;FOLD ARCOFF WDAT2 LIN P4 CPDAT2 Tool[1]:cmttorch Base[1]:vrashatel ;%{PE}
  ;FOLD Parameters ;%{h}
    ;Params IlfProvider=kukaroboter.arctech.arcofflin; Kuka.IsGlobalPoint=False; Kuka.PointName=P4; Kuka.BlendingEnabled=False; Kuka.MoveDataName=CPDAT2; Kuka.VelocityPath=0.01; Kuka.CurrentCDSetIndex=0; Kuka.MovementParameterFieldEnabled=True; ArcTech.WdatVarName=WDAT2; ArcTech.Basic=3.4.3.1264
  ;ENDFOLD
  $BWDSTART = FALSE
  LDAT_ACT = LCPDAT2
  FDAT_ACT = FP4
  BAS(#CP_PARAMS, gArcBasVelDefinition)
  SET_CD_PARAMS (0)
  TRIGGER WHEN PATH = ArcGetPath(#ArcOffBefore, WDAT2) DELAY = 0 DO ArcMainNG(#ArcOffBeforeOffStd, WDAT2, WP4) PRIO = -1
  TRIGGER WHEN PATH = ArcGetPath(#OnTheFlyArcOff, WDAT2) DELAY = 0 DO ArcMainNG(#ArcOffMoveStd, WDAT2, WP4) PRIO = -1
  ArcMainNG(#ArcOffBeforeMoveStd, WDAT2, WP4)
  LIN XP4
  ArcMainNG(#ArcOffAfterMoveStd, WDAT2, WP4)
;ENDFOLD
   $VEL.CP = 0.080
   LIN  {X 8.829, Y -0.910, Z 19.700, A 0.000, B 0.000, C 0.000} C_DIS

;FOLD ARCON WDAT1 LIN P3 Vel=0.5 m/s CPDAT1 Tool[1]:cmttorch Base[1]:vrashatel ;%{PE}
  ;FOLD Parameters ;%{h}
    ;Params IlfProvider=kukaroboter.arctech.arconlin; Kuka.IsGlobalPoint=False; Kuka.PointName=P3; Kuka.BlendingEnabled=False; Kuka.MoveDataName=CPDAT1; Kuka.VelocityPath=0.5; Kuka.CurrentCDSetIndex=0; Kuka.MovementParameterFieldEnabled=True; ArcTech.WdatVarName=WDAT1; ArcTech.Basic=3.4.3.1264
  ;ENDFOLD
  $BWDSTART = FALSE
  LDAT_ACT = LCPDAT1
  FDAT_ACT = FP3
  BAS(#CP_PARAMS, 0.5)
  SET_CD_PARAMS (0)
  TRIGGER WHEN DISTANCE = 1 DELAY = ArcGetDelay(#PreDefinition, WDAT1) DO ArcMainNG(#PreDefinition, WDAT1, WP3) PRIO = -1
  TRIGGER WHEN PATH = ArcGetPath(#OnTheFlyArcOn, WDAT1) DELAY = ArcGetDelay(#GasPreflow, WDAT1) DO ArcMainNG(#GasPreflow, WDAT1, WP3) PRIO = -1
  TRIGGER WHEN PATH = ArcGetPath(#OnTheFlyArcOn, WDAT1) DELAY = 0 DO ArcMainNG(#ArcOnMoveStd, WDAT1, WP3) PRIO = -1
  ArcMainNG(#ArcOnBeforeMoveStd, WDAT1, WP3)
  LIN XP3
  ArcMainNG(#ArcOnAfterMoveStd, WDAT1, WP3)
;ENDFOLD
   $VEL.CP = 0.060
   LIN  {X 4.151, Y 3.768, Z 19.700, A 0.000, B 0.000, C 0.000} C_DIS

;FOLD ARCOFF WDAT2 LIN P4 CPDAT2 Tool[1]:cmttorch Base[1]:vrashatel ;%{PE}
  ;FOLD Parameters ;%{h}
    ;Params IlfProvider=kukaroboter.arctech.arcofflin; Kuka.IsGlobalPoint=False; Kuka.PointName=P4; Kuka.BlendingEnabled=False; Kuka.MoveDataName=CPDAT2; Kuka.VelocityPath=0.01; Kuka.CurrentCDSetIndex=0; Kuka.MovementParameterFieldEnabled=True; ArcTech.WdatVarName=WDAT2; ArcTech.Basic=3.4.3.1264
  ;ENDFOLD
  $BWDSTART = FALSE
  LDAT_ACT = LCPDAT2
  FDAT_ACT = FP4
  BAS(#CP_PARAMS, gArcBasVelDefinition)
  SET_CD_PARAMS (0)
  TRIGGER WHEN PATH = ArcGetPath(#ArcOffBefore, WDAT2) DELAY = 0 DO ArcMainNG(#ArcOffBeforeOffStd, WDAT2, WP4) PRIO = -1
  TRIGGER WHEN PATH = ArcGetPath(#OnTheFlyArcOff, WDAT2) DELAY = 0 DO ArcMainNG(#ArcOffMoveStd, WDAT2, WP4) PRIO = -1
  ArcMainNG(#ArcOffBeforeMoveStd, WDAT2, WP4)
  LIN XP4
  ArcMainNG(#ArcOffAfterMoveStd, WDAT2, WP4)
;ENDFOLD
   $VEL.CP = 0.080
   LIN  {X 4.343, Y 4.142, Z 19.700, A 0.000, B 0.000, C 0.000} C_DIS

;FOLD ARCON WDAT1 LIN P3 Vel=0.5 m/s CPDAT1 Tool[1]:cmttorch Base[1]:vrashatel ;%{PE}
  ;FOLD Parameters ;%{h}
    ;Params IlfProvider=kukaroboter.arctech.arconlin; Kuka.IsGlobalPoint=False; Kuka.PointName=P3; Kuka.BlendingEnabled=False; Kuka.MoveDataName=CPDAT1; Kuka.VelocityPath=0.5; Kuka.CurrentCDSetIndex=0; Kuka.MovementParameterFieldEnabled=True; ArcTech.WdatVarName=WDAT1; ArcTech.Basic=3.4.3.1264
  ;ENDFOLD
  $BWDSTART = FALSE
  LDAT_ACT = LCPDAT1
  FDAT_ACT = FP3
  BAS(#CP_PARAMS, 0.5)
  SET_CD_PARAMS (0)
  TRIGGER WHEN DISTANCE = 1 DELAY = ArcGetDelay(#PreDefinition, WDAT1) DO ArcMainNG(#PreDefinition, WDAT1, WP3) PRIO = -1
  TRIGGER WHEN PATH = ArcGetPath(#OnTheFlyArcOn, WDAT1) DELAY = ArcGetDelay(#GasPreflow, WDAT1) DO ArcMainNG(#GasPreflow, WDAT1, WP3) PRIO = -1
  TRIGGER WHEN PATH = ArcGetPath(#OnTheFlyArcOn, WDAT1) DELAY = 0 DO ArcMainNG(#ArcOnMoveStd, WDAT1, WP3) PRIO = -1
  ArcMainNG(#ArcOnBeforeMoveStd, WDAT1, WP3)
  LIN XP3
  ArcMainNG(#ArcOnAfterMoveStd, WDAT1, WP3)
;ENDFOLD
   $VEL.CP = 0.060
   LIN  {X 8.829, Y -0.344, Z 19.700, A 0.000, B 0.000, C 0.000} C_DIS

;FOLD ARCOFF WDAT2 LIN P4 CPDAT2 Tool[1]:cmttorch Base[1]:vrashatel ;%{PE}
  ;FOLD Parameters ;%{h}
    ;Params IlfProvider=kukaroboter.arctech.arcofflin; Kuka.IsGlobalPoint=False; Kuka.PointName=P4; Kuka.BlendingEnabled=False; Kuka.MoveDataName=CPDAT2; Kuka.VelocityPath=0.01; Kuka.CurrentCDSetIndex=0; Kuka.MovementParameterFieldEnabled=True; ArcTech.WdatVarName=WDAT2; ArcTech.Basic=3.4.3.1264
  ;ENDFOLD
  $BWDSTART = FALSE
  LDAT_ACT = LCPDAT2
  FDAT_ACT = FP4
  BAS(#CP_PARAMS, gArcBasVelDefinition)
  SET_CD_PARAMS (0)
  TRIGGER WHEN PATH = ArcGetPath(#ArcOffBefore, WDAT2) DELAY = 0 DO ArcMainNG(#ArcOffBeforeOffStd, WDAT2, WP4) PRIO = -1
  TRIGGER WHEN PATH = ArcGetPath(#OnTheFlyArcOff, WDAT2) DELAY = 0 DO ArcMainNG(#ArcOffMoveStd, WDAT2, WP4) PRIO = -1
  ArcMainNG(#ArcOffBeforeMoveStd, WDAT2, WP4)
  LIN XP4
  ArcMainNG(#ArcOffAfterMoveStd, WDAT2, WP4)
;ENDFOLD
   $VEL.CP = 0.080
   LIN  {X 8.829, Y 0.221, Z 19.700, A 0.000, B 0.000, C 0.000} C_DIS

;FOLD ARCON WDAT1 LIN P3 Vel=0.5 m/s CPDAT1 Tool[1]:cmttorch Base[1]:vrashatel ;%{PE}
  ;FOLD Parameters ;%{h}
    ;Params IlfProvider=kukaroboter.arctech.arconlin; Kuka.IsGlobalPoint=False; Kuka.PointName=P3; Kuka.BlendingEnabled=False; Kuka.MoveDataName=CPDAT1; Kuka.VelocityPath=0.5; Kuka.CurrentCDSetIndex=0; Kuka.MovementParameterFieldEnabled=True; ArcTech.WdatVarName=WDAT1; ArcTech.Basic=3.4.3.1264
  ;ENDFOLD
  $BWDSTART = FALSE
  LDAT_ACT = LCPDAT1
  FDAT_ACT = FP3
  BAS(#CP_PARAMS, 0.5)
  SET_CD_PARAMS (0)
  TRIGGER WHEN DISTANCE = 1 DELAY = ArcGetDelay(#PreDefinition, WDAT1) DO ArcMainNG(#PreDefinition, WDAT1, WP3) PRIO = -1
  TRIGGER WHEN PATH = ArcGetPath(#OnTheFlyArcOn, WDAT1) DELAY = ArcGetDelay(#GasPreflow, WDAT1) DO ArcMainNG(#GasPreflow, WDAT1, WP3) PRIO = -1
  TRIGGER WHEN PATH = ArcGetPath(#OnTheFlyArcOn, WDAT1) DELAY = 0 DO ArcMainNG(#ArcOnMoveStd, WDAT1, WP3) PRIO = -1
  ArcMainNG(#ArcOnBeforeMoveStd, WDAT1, WP3)
  LIN XP3
  ArcMainNG(#ArcOnAfterMoveStd, WDAT1, WP3)
;ENDFOLD
   $VEL.CP = 0.060
   LIN  {X 4.534, Y 4.516, Z 19.700, A 0.000, B 0.000, C 0.000} C_DIS

;FOLD ARCOFF WDAT2 LIN P4 CPDAT2 Tool[1]:cmttorch Base[1]:vrashatel ;%{PE}
  ;FOLD Parameters ;%{h}
    ;Params IlfProvider=kukaroboter.arctech.arcofflin; Kuka.IsGlobalPoint=False; Kuka.PointName=P4; Kuka.BlendingEnabled=False; Kuka.MoveDataName=CPDAT2; Kuka.VelocityPath=0.01; Kuka.CurrentCDSetIndex=0; Kuka.MovementParameterFieldEnabled=True; ArcTech.WdatVarName=WDAT2; ArcTech.Basic=3.4.3.1264
  ;ENDFOLD
  $BWDSTART = FALSE
  LDAT_ACT = LCPDAT2
  FDAT_ACT = FP4
  BAS(#CP_PARAMS, gArcBasVelDefinition)
  SET_CD_PARAMS (0)
  TRIGGER WHEN PATH = ArcGetPath(#ArcOffBefore, WDAT2) DELAY = 0 DO ArcMainNG(#ArcOffBeforeOffStd, WDAT2, WP4) PRIO = -1
  TRIGGER WHEN PATH = ArcGetPath(#OnTheFlyArcOff, WDAT2) DELAY = 0 DO ArcMainNG(#ArcOffMoveStd, WDAT2, WP4) PRIO = -1
  ArcMainNG(#ArcOffBeforeMoveStd, WDAT2, WP4)
  LIN XP4
  ArcMainNG(#ArcOffAfterMoveStd, WDAT2, WP4)
;ENDFOLD
   $VEL.CP = 0.080
   LIN  {X 4.726, Y 4.890, Z 19.700, A 0.000, B 0.000, C 0.000} C_DIS

;FOLD ARCON WDAT1 LIN P3 Vel=0.5 m/s CPDAT1 Tool[1]:cmttorch Base[1]:vrashatel ;%{PE}
  ;FOLD Parameters ;%{h}
    ;Params IlfProvider=kukaroboter.arctech.arconlin; Kuka.IsGlobalPoint=False; Kuka.PointName=P3; Kuka.BlendingEnabled=False; Kuka.MoveDataName=CPDAT1; Kuka.VelocityPath=0.5; Kuka.CurrentCDSetIndex=0; Kuka.MovementParameterFieldEnabled=True; ArcTech.WdatVarName=WDAT1; ArcTech.Basic=3.4.3.1264
  ;ENDFOLD
  $BWDSTART = FALSE
  LDAT_ACT = LCPDAT1
  FDAT_ACT = FP3
  BAS(#CP_PARAMS, 0.5)
  SET_CD_PARAMS (0)
  TRIGGER WHEN DISTANCE = 1 DELAY = ArcGetDelay(#PreDefinition, WDAT1) DO ArcMainNG(#PreDefinition, WDAT1, WP3) PRIO = -1
  TRIGGER WHEN PATH = ArcGetPath(#OnTheFlyArcOn, WDAT1) DELAY = ArcGetDelay(#GasPreflow, WDAT1) DO ArcMainNG(#GasPreflow, WDAT1, WP3) PRIO = -1
  TRIGGER WHEN PATH = ArcGetPath(#OnTheFlyArcOn, WDAT1) DELAY = 0 DO ArcMainNG(#ArcOnMoveStd, WDAT1, WP3) PRIO = -1
  ArcMainNG(#ArcOnBeforeMoveStd, WDAT1, WP3)
  LIN XP3
  ArcMainNG(#ArcOnAfterMoveStd, WDAT1, WP3)
;ENDFOLD
   $VEL.CP = 0.060
   LIN  {X 8.829, Y 0.787, Z 19.700, A 0.000, B 0.000, C 0.000} C_DIS

;FOLD ARCOFF WDAT2 LIN P4 CPDAT2 Tool[1]:cmttorch Base[1]:vrashatel ;%{PE}
  ;FOLD Parameters ;%{h}
    ;Params IlfProvider=kukaroboter.arctech.arcofflin; Kuka.IsGlobalPoint=False; Kuka.PointName=P4; Kuka.BlendingEnabled=False; Kuka.MoveDataName=CPDAT2; Kuka.VelocityPath=0.01; Kuka.CurrentCDSetIndex=0; Kuka.MovementParameterFieldEnabled=True; ArcTech.WdatVarName=WDAT2; ArcTech.Basic=3.4.3.1264
  ;ENDFOLD
  $BWDSTART = FALSE
  LDAT_ACT = LCPDAT2
  FDAT_ACT = FP4
  BAS(#CP_PARAMS, gArcBasVelDefinition)
  SET_CD_PARAMS (0)
  TRIGGER WHEN PATH = ArcGetPath(#ArcOffBefore, WDAT2) DELAY = 0 DO ArcMainNG(#ArcOffBeforeOffStd, WDAT2, WP4) PRIO = -1
  TRIGGER WHEN PATH = ArcGetPath(#OnTheFlyArcOff, WDAT2) DELAY = 0 DO ArcMainNG(#ArcOffMoveStd, WDAT2, WP4) PRIO = -1
  ArcMainNG(#ArcOffBeforeMoveStd, WDAT2, WP4)
  LIN XP4
  ArcMainNG(#ArcOffAfterMoveStd, WDAT2, WP4)
;ENDFOLD
   $VEL.CP = 0.080
   LIN  {X 8.829, Y 1.352, Z 19.700, A 0.000, B 0.000, C 0.000} C_DIS

;FOLD ARCON WDAT1 LIN P3 Vel=0.5 m/s CPDAT1 Tool[1]:cmttorch Base[1]:vrashatel ;%{PE}
  ;FOLD Parameters ;%{h}
    ;Params IlfProvider=kukaroboter.arctech.arconlin; Kuka.IsGlobalPoint=False; Kuka.PointName=P3; Kuka.BlendingEnabled=False; Kuka.MoveDataName=CPDAT1; Kuka.VelocityPath=0.5; Kuka.CurrentCDSetIndex=0; Kuka.MovementParameterFieldEnabled=True; ArcTech.WdatVarName=WDAT1; ArcTech.Basic=3.4.3.1264
  ;ENDFOLD
  $BWDSTART = FALSE
  LDAT_ACT = LCPDAT1
  FDAT_ACT = FP3
  BAS(#CP_PARAMS, 0.5)
  SET_CD_PARAMS (0)
  TRIGGER WHEN DISTANCE = 1 DELAY = ArcGetDelay(#PreDefinition, WDAT1) DO ArcMainNG(#PreDefinition, WDAT1, WP3) PRIO = -1
  TRIGGER WHEN PATH = ArcGetPath(#OnTheFlyArcOn, WDAT1) DELAY = ArcGetDelay(#GasPreflow, WDAT1) DO ArcMainNG(#GasPreflow, WDAT1, WP3) PRIO = -1
  TRIGGER WHEN PATH = ArcGetPath(#OnTheFlyArcOn, WDAT1) DELAY = 0 DO ArcMainNG(#ArcOnMoveStd, WDAT1, WP3) PRIO = -1
  ArcMainNG(#ArcOnBeforeMoveStd, WDAT1, WP3)
  LIN XP3
  ArcMainNG(#ArcOnAfterMoveStd, WDAT1, WP3)
;ENDFOLD
   $VEL.CP = 0.060
   LIN  {X 4.917, Y 5.264, Z 19.700, A 0.000, B 0.000, C 0.000} C_DIS

;FOLD ARCOFF WDAT2 LIN P4 CPDAT2 Tool[1]:cmttorch Base[1]:vrashatel ;%{PE}
  ;FOLD Parameters ;%{h}
    ;Params IlfProvider=kukaroboter.arctech.arcofflin; Kuka.IsGlobalPoint=False; Kuka.PointName=P4; Kuka.BlendingEnabled=False; Kuka.MoveDataName=CPDAT2; Kuka.VelocityPath=0.01; Kuka.CurrentCDSetIndex=0; Kuka.MovementParameterFieldEnabled=True; ArcTech.WdatVarName=WDAT2; ArcTech.Basic=3.4.3.1264
  ;ENDFOLD
  $BWDSTART = FALSE
  LDAT_ACT = LCPDAT2
  FDAT_ACT = FP4
  BAS(#CP_PARAMS, gArcBasVelDefinition)
  SET_CD_PARAMS (0)
  TRIGGER WHEN PATH = ArcGetPath(#ArcOffBefore, WDAT2) DELAY = 0 DO ArcMainNG(#ArcOffBeforeOffStd, WDAT2, WP4) PRIO = -1
  TRIGGER WHEN PATH = ArcGetPath(#OnTheFlyArcOff, WDAT2) DELAY = 0 DO ArcMainNG(#ArcOffMoveStd, WDAT2, WP4) PRIO = -1
  ArcMainNG(#ArcOffBeforeMoveStd, WDAT2, WP4)
  LIN XP4
  ArcMainNG(#ArcOffAfterMoveStd, WDAT2, WP4)
;ENDFOLD
   $VEL.CP = 0.080
   LIN  {X 5.096, Y 5.651, Z 19.700, A 0.000, B 0.000, C 0.000} C_DIS

;FOLD ARCON WDAT1 LIN P3 Vel=0.5 m/s CPDAT1 Tool[1]:cmttorch Base[1]:vrashatel ;%{PE}
  ;FOLD Parameters ;%{h}
    ;Params IlfProvider=kukaroboter.arctech.arconlin; Kuka.IsGlobalPoint=False; Kuka.PointName=P3; Kuka.BlendingEnabled=False; Kuka.MoveDataName=CPDAT1; Kuka.VelocityPath=0.5; Kuka.CurrentCDSetIndex=0; Kuka.MovementParameterFieldEnabled=True; ArcTech.WdatVarName=WDAT1; ArcTech.Basic=3.4.3.1264
  ;ENDFOLD
  $BWDSTART = FALSE
  LDAT_ACT = LCPDAT1
  FDAT_ACT = FP3
  BAS(#CP_PARAMS, 0.5)
  SET_CD_PARAMS (0)
  TRIGGER WHEN DISTANCE = 1 DELAY = ArcGetDelay(#PreDefinition, WDAT1) DO ArcMainNG(#PreDefinition, WDAT1, WP3) PRIO = -1
  TRIGGER WHEN PATH = ArcGetPath(#OnTheFlyArcOn, WDAT1) DELAY = ArcGetDelay(#GasPreflow, WDAT1) DO ArcMainNG(#GasPreflow, WDAT1, WP3) PRIO = -1
  TRIGGER WHEN PATH = ArcGetPath(#OnTheFlyArcOn, WDAT1) DELAY = 0 DO ArcMainNG(#ArcOnMoveStd, WDAT1, WP3) PRIO = -1
  ArcMainNG(#ArcOnBeforeMoveStd, WDAT1, WP3)
  LIN XP3
  ArcMainNG(#ArcOnAfterMoveStd, WDAT1, WP3)
;ENDFOLD
   $VEL.CP = 0.060
   LIN  {X 8.829, Y 1.918, Z 19.700, A 0.000, B 0.000, C 0.000} C_DIS

;FOLD ARCOFF WDAT2 LIN P4 CPDAT2 Tool[1]:cmttorch Base[1]:vrashatel ;%{PE}
  ;FOLD Parameters ;%{h}
    ;Params IlfProvider=kukaroboter.arctech.arcofflin; Kuka.IsGlobalPoint=False; Kuka.PointName=P4; Kuka.BlendingEnabled=False; Kuka.MoveDataName=CPDAT2; Kuka.VelocityPath=0.01; Kuka.CurrentCDSetIndex=0; Kuka.MovementParameterFieldEnabled=True; ArcTech.WdatVarName=WDAT2; ArcTech.Basic=3.4.3.1264
  ;ENDFOLD
  $BWDSTART = FALSE
  LDAT_ACT = LCPDAT2
  FDAT_ACT = FP4
  BAS(#CP_PARAMS, gArcBasVelDefinition)
  SET_CD_PARAMS (0)
  TRIGGER WHEN PATH = ArcGetPath(#ArcOffBefore, WDAT2) DELAY = 0 DO ArcMainNG(#ArcOffBeforeOffStd, WDAT2, WP4) PRIO = -1
  TRIGGER WHEN PATH = ArcGetPath(#OnTheFlyArcOff, WDAT2) DELAY = 0 DO ArcMainNG(#ArcOffMoveStd, WDAT2, WP4) PRIO = -1
  ArcMainNG(#ArcOffBeforeMoveStd, WDAT2, WP4)
  LIN XP4
  ArcMainNG(#ArcOffAfterMoveStd, WDAT2, WP4)
;ENDFOLD
   $VEL.CP = 0.080
   LIN  {X 8.829, Y 2.484, Z 19.700, A 0.000, B 0.000, C 0.000} C_DIS

;FOLD ARCON WDAT1 LIN P3 Vel=0.5 m/s CPDAT1 Tool[1]:cmttorch Base[1]:vrashatel ;%{PE}
  ;FOLD Parameters ;%{h}
    ;Params IlfProvider=kukaroboter.arctech.arconlin; Kuka.IsGlobalPoint=False; Kuka.PointName=P3; Kuka.BlendingEnabled=False; Kuka.MoveDataName=CPDAT1; Kuka.VelocityPath=0.5; Kuka.CurrentCDSetIndex=0; Kuka.MovementParameterFieldEnabled=True; ArcTech.WdatVarName=WDAT1; ArcTech.Basic=3.4.3.1264
  ;ENDFOLD
  $BWDSTART = FALSE
  LDAT_ACT = LCPDAT1
  FDAT_ACT = FP3
  BAS(#CP_PARAMS, 0.5)
  SET_CD_PARAMS (0)
  TRIGGER WHEN DISTANCE = 1 DELAY = ArcGetDelay(#PreDefinition, WDAT1) DO ArcMainNG(#PreDefinition, WDAT1, WP3) PRIO = -1
  TRIGGER WHEN PATH = ArcGetPath(#OnTheFlyArcOn, WDAT1) DELAY = ArcGetDelay(#GasPreflow, WDAT1) DO ArcMainNG(#GasPreflow, WDAT1, WP3) PRIO = -1
  TRIGGER WHEN PATH = ArcGetPath(#OnTheFlyArcOn, WDAT1) DELAY = 0 DO ArcMainNG(#ArcOnMoveStd, WDAT1, WP3) PRIO = -1
  ArcMainNG(#ArcOnBeforeMoveStd, WDAT1, WP3)
  LIN XP3
  ArcMainNG(#ArcOnAfterMoveStd, WDAT1, WP3)
;ENDFOLD
   $VEL.CP = 0.060
   LIN  {X 5.096, Y 6.216, Z 19.700, A 0.000, B 0.000, C 0.000} C_DIS

;FOLD ARCOFF WDAT2 LIN P4 CPDAT2 Tool[1]:cmttorch Base[1]:vrashatel ;%{PE}
  ;FOLD Parameters ;%{h}
    ;Params IlfProvider=kukaroboter.arctech.arcofflin; Kuka.IsGlobalPoint=False; Kuka.PointName=P4; Kuka.BlendingEnabled=False; Kuka.MoveDataName=CPDAT2; Kuka.VelocityPath=0.01; Kuka.CurrentCDSetIndex=0; Kuka.MovementParameterFieldEnabled=True; ArcTech.WdatVarName=WDAT2; ArcTech.Basic=3.4.3.1264
  ;ENDFOLD
  $BWDSTART = FALSE
  LDAT_ACT = LCPDAT2
  FDAT_ACT = FP4
  BAS(#CP_PARAMS, gArcBasVelDefinition)
  SET_CD_PARAMS (0)
  TRIGGER WHEN PATH = ArcGetPath(#ArcOffBefore, WDAT2) DELAY = 0 DO ArcMainNG(#ArcOffBeforeOffStd, WDAT2, WP4) PRIO = -1
  TRIGGER WHEN PATH = ArcGetPath(#OnTheFlyArcOff, WDAT2) DELAY = 0 DO ArcMainNG(#ArcOffMoveStd, WDAT2, WP4) PRIO = -1
  ArcMainNG(#ArcOffBeforeMoveStd, WDAT2, WP4)
  LIN XP4
  ArcMainNG(#ArcOffAfterMoveStd, WDAT2, WP4)
;ENDFOLD
   $VEL.CP = 0.080
   LIN  {X 5.096, Y 6.782, Z 19.700, A 0.000, B 0.000, C 0.000} C_DIS

;FOLD ARCON WDAT1 LIN P3 Vel=0.5 m/s CPDAT1 Tool[1]:cmttorch Base[1]:vrashatel ;%{PE}
  ;FOLD Parameters ;%{h}
    ;Params IlfProvider=kukaroboter.arctech.arconlin; Kuka.IsGlobalPoint=False; Kuka.PointName=P3; Kuka.BlendingEnabled=False; Kuka.MoveDataName=CPDAT1; Kuka.VelocityPath=0.5; Kuka.CurrentCDSetIndex=0; Kuka.MovementParameterFieldEnabled=True; ArcTech.WdatVarName=WDAT1; ArcTech.Basic=3.4.3.1264
  ;ENDFOLD
  $BWDSTART = FALSE
  LDAT_ACT = LCPDAT1
  FDAT_ACT = FP3
  BAS(#CP_PARAMS, 0.5)
  SET_CD_PARAMS (0)
  TRIGGER WHEN DISTANCE = 1 DELAY = ArcGetDelay(#PreDefinition, WDAT1) DO ArcMainNG(#PreDefinition, WDAT1, WP3) PRIO = -1
  TRIGGER WHEN PATH = ArcGetPath(#OnTheFlyArcOn, WDAT1) DELAY = ArcGetDelay(#GasPreflow, WDAT1) DO ArcMainNG(#GasPreflow, WDAT1, WP3) PRIO = -1
  TRIGGER WHEN PATH = ArcGetPath(#OnTheFlyArcOn, WDAT1) DELAY = 0 DO ArcMainNG(#ArcOnMoveStd, WDAT1, WP3) PRIO = -1
  ArcMainNG(#ArcOnBeforeMoveStd, WDAT1, WP3)
  LIN XP3
  ArcMainNG(#ArcOnAfterMoveStd, WDAT1, WP3)
;ENDFOLD
   $VEL.CP = 0.060
   LIN  {X 8.829, Y 3.049, Z 19.700, A 0.000, B 0.000, C 0.000} C_DIS

;FOLD ARCOFF WDAT2 LIN P4 CPDAT2 Tool[1]:cmttorch Base[1]:vrashatel ;%{PE}
  ;FOLD Parameters ;%{h}
    ;Params IlfProvider=kukaroboter.arctech.arcofflin; Kuka.IsGlobalPoint=False; Kuka.PointName=P4; Kuka.BlendingEnabled=False; Kuka.MoveDataName=CPDAT2; Kuka.VelocityPath=0.01; Kuka.CurrentCDSetIndex=0; Kuka.MovementParameterFieldEnabled=True; ArcTech.WdatVarName=WDAT2; ArcTech.Basic=3.4.3.1264
  ;ENDFOLD
  $BWDSTART = FALSE
  LDAT_ACT = LCPDAT2
  FDAT_ACT = FP4
  BAS(#CP_PARAMS, gArcBasVelDefinition)
  SET_CD_PARAMS (0)
  TRIGGER WHEN PATH = ArcGetPath(#ArcOffBefore, WDAT2) DELAY = 0 DO ArcMainNG(#ArcOffBeforeOffStd, WDAT2, WP4) PRIO = -1
  TRIGGER WHEN PATH = ArcGetPath(#OnTheFlyArcOff, WDAT2) DELAY = 0 DO ArcMainNG(#ArcOffMoveStd, WDAT2, WP4) PRIO = -1
  ArcMainNG(#ArcOffBeforeMoveStd, WDAT2, WP4)
  LIN XP4
  ArcMainNG(#ArcOffAfterMoveStd, WDAT2, WP4)
;ENDFOLD
   $VEL.CP = 0.060
   LIN  {X 8.899, Y 2.979, Z 19.700, A 0.000, B 0.000, C 0.000} C_DIS
   $VEL.CP = 0.080
   LIN  {X 9.290, Y 2.979, Z 19.700, A 0.000, B 0.000, C 0.000} C_DIS
   $VEL.CP = 0.080
   LIN  {X 9.218, Y -9.218, Z 19.700, A 0.000, B 0.000, C 0.000} C_DIS
   $VEL.CP = 0.080
   LIN  {X -3.615, Y -9.290, Z 19.700, A 0.000, B 0.000, C 0.000} C_DIS
   $VEL.CP = 0.080
   LIN  {X -3.615, Y -8.829, Z 19.700, A 0.000, B 0.000, C 0.000} C_DIS

;FOLD ARCON WDAT1 LIN P3 Vel=0.5 m/s CPDAT1 Tool[1]:cmttorch Base[1]:vrashatel ;%{PE}
  ;FOLD Parameters ;%{h}
    ;Params IlfProvider=kukaroboter.arctech.arconlin; Kuka.IsGlobalPoint=False; Kuka.PointName=P3; Kuka.BlendingEnabled=False; Kuka.MoveDataName=CPDAT1; Kuka.VelocityPath=0.5; Kuka.CurrentCDSetIndex=0; Kuka.MovementParameterFieldEnabled=True; ArcTech.WdatVarName=WDAT1; ArcTech.Basic=3.4.3.1264
  ;ENDFOLD
  $BWDSTART = FALSE
  LDAT_ACT = LCPDAT1
  FDAT_ACT = FP3
  BAS(#CP_PARAMS, 0.5)
  SET_CD_PARAMS (0)
  TRIGGER WHEN DISTANCE = 1 DELAY = ArcGetDelay(#PreDefinition, WDAT1) DO ArcMainNG(#PreDefinition, WDAT1, WP3) PRIO = -1
  TRIGGER WHEN PATH = ArcGetPath(#OnTheFlyArcOn, WDAT1) DELAY = ArcGetDelay(#GasPreflow, WDAT1) DO ArcMainNG(#GasPreflow, WDAT1, WP3) PRIO = -1
  TRIGGER WHEN PATH = ArcGetPath(#OnTheFlyArcOn, WDAT1) DELAY = 0 DO ArcMainNG(#ArcOnMoveStd, WDAT1, WP3) PRIO = -1
  ArcMainNG(#ArcOnBeforeMoveStd, WDAT1, WP3)
  LIN XP3
  ArcMainNG(#ArcOnAfterMoveStd, WDAT1, WP3)
;ENDFOLD
   $VEL.CP = 0.025
   LIN  {X -3.615, Y -8.829, Z 19.700, A 0.000, B 0.000, C 0.000} C_DIS
   $VEL.CP = 0.060
   LIN  {X -8.829, Y -3.615, Z 19.700, A 0.000, B 0.000, C 0.000} C_DIS

;FOLD ARCOFF WDAT2 LIN P4 CPDAT2 Tool[1]:cmttorch Base[1]:vrashatel ;%{PE}
  ;FOLD Parameters ;%{h}
    ;Params IlfProvider=kukaroboter.arctech.arcofflin; Kuka.IsGlobalPoint=False; Kuka.PointName=P4; Kuka.BlendingEnabled=False; Kuka.MoveDataName=CPDAT2; Kuka.VelocityPath=0.01; Kuka.CurrentCDSetIndex=0; Kuka.MovementParameterFieldEnabled=True; ArcTech.WdatVarName=WDAT2; ArcTech.Basic=3.4.3.1264
  ;ENDFOLD
  $BWDSTART = FALSE
  LDAT_ACT = LCPDAT2
  FDAT_ACT = FP4
  BAS(#CP_PARAMS, gArcBasVelDefinition)
  SET_CD_PARAMS (0)
  TRIGGER WHEN PATH = ArcGetPath(#ArcOffBefore, WDAT2) DELAY = 0 DO ArcMainNG(#ArcOffBeforeOffStd, WDAT2, WP4) PRIO = -1
  TRIGGER WHEN PATH = ArcGetPath(#OnTheFlyArcOff, WDAT2) DELAY = 0 DO ArcMainNG(#ArcOffMoveStd, WDAT2, WP4) PRIO = -1
  ArcMainNG(#ArcOffBeforeMoveStd, WDAT2, WP4)
  LIN XP4
  ArcMainNG(#ArcOffAfterMoveStd, WDAT2, WP4)
;ENDFOLD
   $VEL.CP = 0.080
   LIN  {X -8.829, Y -4.181, Z 19.700, A 0.000, B 0.000, C 0.000} C_DIS

;FOLD ARCON WDAT1 LIN P3 Vel=0.5 m/s CPDAT1 Tool[1]:cmttorch Base[1]:vrashatel ;%{PE}
  ;FOLD Parameters ;%{h}
    ;Params IlfProvider=kukaroboter.arctech.arconlin; Kuka.IsGlobalPoint=False; Kuka.PointName=P3; Kuka.BlendingEnabled=False; Kuka.MoveDataName=CPDAT1; Kuka.VelocityPath=0.5; Kuka.CurrentCDSetIndex=0; Kuka.MovementParameterFieldEnabled=True; ArcTech.WdatVarName=WDAT1; ArcTech.Basic=3.4.3.1264
  ;ENDFOLD
  $BWDSTART = FALSE
  LDAT_ACT = LCPDAT1
  FDAT_ACT = FP3
  BAS(#CP_PARAMS, 0.5)
  SET_CD_PARAMS (0)
  TRIGGER WHEN DISTANCE = 1 DELAY = ArcGetDelay(#PreDefinition, WDAT1) DO ArcMainNG(#PreDefinition, WDAT1, WP3) PRIO = -1
  TRIGGER WHEN PATH = ArcGetPath(#OnTheFlyArcOn, WDAT1) DELAY = ArcGetDelay(#GasPreflow, WDAT1) DO ArcMainNG(#GasPreflow, WDAT1, WP3) PRIO = -1
  TRIGGER WHEN PATH = ArcGetPath(#OnTheFlyArcOn, WDAT1) DELAY = 0 DO ArcMainNG(#ArcOnMoveStd, WDAT1, WP3) PRIO = -1
  ArcMainNG(#ArcOnBeforeMoveStd, WDAT1, WP3)
  LIN XP3
  ArcMainNG(#ArcOnAfterMoveStd, WDAT1, WP3)
;ENDFOLD
   $VEL.CP = 0.060
   LIN  {X -4.181, Y -8.829, Z 19.700, A 0.000, B 0.000, C 0.000} C_DIS

;FOLD ARCOFF WDAT2 LIN P4 CPDAT2 Tool[1]:cmttorch Base[1]:vrashatel ;%{PE}
  ;FOLD Parameters ;%{h}
    ;Params IlfProvider=kukaroboter.arctech.arcofflin; Kuka.IsGlobalPoint=False; Kuka.PointName=P4; Kuka.BlendingEnabled=False; Kuka.MoveDataName=CPDAT2; Kuka.VelocityPath=0.01; Kuka.CurrentCDSetIndex=0; Kuka.MovementParameterFieldEnabled=True; ArcTech.WdatVarName=WDAT2; ArcTech.Basic=3.4.3.1264
  ;ENDFOLD
  $BWDSTART = FALSE
  LDAT_ACT = LCPDAT2
  FDAT_ACT = FP4
  BAS(#CP_PARAMS, gArcBasVelDefinition)
  SET_CD_PARAMS (0)
  TRIGGER WHEN PATH = ArcGetPath(#ArcOffBefore, WDAT2) DELAY = 0 DO ArcMainNG(#ArcOffBeforeOffStd, WDAT2, WP4) PRIO = -1
  TRIGGER WHEN PATH = ArcGetPath(#OnTheFlyArcOff, WDAT2) DELAY = 0 DO ArcMainNG(#ArcOffMoveStd, WDAT2, WP4) PRIO = -1
  ArcMainNG(#ArcOffBeforeMoveStd, WDAT2, WP4)
  LIN XP4
  ArcMainNG(#ArcOffAfterMoveStd, WDAT2, WP4)
;ENDFOLD
   $VEL.CP = 0.080
   LIN  {X -4.746, Y -8.829, Z 19.700, A 0.000, B 0.000, C 0.000} C_DIS

;FOLD ARCON WDAT1 LIN P3 Vel=0.5 m/s CPDAT1 Tool[1]:cmttorch Base[1]:vrashatel ;%{PE}
  ;FOLD Parameters ;%{h}
    ;Params IlfProvider=kukaroboter.arctech.arconlin; Kuka.IsGlobalPoint=False; Kuka.PointName=P3; Kuka.BlendingEnabled=False; Kuka.MoveDataName=CPDAT1; Kuka.VelocityPath=0.5; Kuka.CurrentCDSetIndex=0; Kuka.MovementParameterFieldEnabled=True; ArcTech.WdatVarName=WDAT1; ArcTech.Basic=3.4.3.1264
  ;ENDFOLD
  $BWDSTART = FALSE
  LDAT_ACT = LCPDAT1
  FDAT_ACT = FP3
  BAS(#CP_PARAMS, 0.5)
  SET_CD_PARAMS (0)
  TRIGGER WHEN DISTANCE = 1 DELAY = ArcGetDelay(#PreDefinition, WDAT1) DO ArcMainNG(#PreDefinition, WDAT1, WP3) PRIO = -1
  TRIGGER WHEN PATH = ArcGetPath(#OnTheFlyArcOn, WDAT1) DELAY = ArcGetDelay(#GasPreflow, WDAT1) DO ArcMainNG(#GasPreflow, WDAT1, WP3) PRIO = -1
  TRIGGER WHEN PATH = ArcGetPath(#OnTheFlyArcOn, WDAT1) DELAY = 0 DO ArcMainNG(#ArcOnMoveStd, WDAT1, WP3) PRIO = -1
  ArcMainNG(#ArcOnBeforeMoveStd, WDAT1, WP3)
  LIN XP3
  ArcMainNG(#ArcOnAfterMoveStd, WDAT1, WP3)
;ENDFOLD
   $VEL.CP = 0.060
   LIN  {X -8.829, Y -4.746, Z 19.700, A 0.000, B 0.000, C 0.000} C_DIS

;FOLD ARCOFF WDAT2 LIN P4 CPDAT2 Tool[1]:cmttorch Base[1]:vrashatel ;%{PE}
  ;FOLD Parameters ;%{h}
    ;Params IlfProvider=kukaroboter.arctech.arcofflin; Kuka.IsGlobalPoint=False; Kuka.PointName=P4; Kuka.BlendingEnabled=False; Kuka.MoveDataName=CPDAT2; Kuka.VelocityPath=0.01; Kuka.CurrentCDSetIndex=0; Kuka.MovementParameterFieldEnabled=True; ArcTech.WdatVarName=WDAT2; ArcTech.Basic=3.4.3.1264
  ;ENDFOLD
  $BWDSTART = FALSE
  LDAT_ACT = LCPDAT2
  FDAT_ACT = FP4
  BAS(#CP_PARAMS, gArcBasVelDefinition)
  SET_CD_PARAMS (0)
  TRIGGER WHEN PATH = ArcGetPath(#ArcOffBefore, WDAT2) DELAY = 0 DO ArcMainNG(#ArcOffBeforeOffStd, WDAT2, WP4) PRIO = -1
  TRIGGER WHEN PATH = ArcGetPath(#OnTheFlyArcOff, WDAT2) DELAY = 0 DO ArcMainNG(#ArcOffMoveStd, WDAT2, WP4) PRIO = -1
  ArcMainNG(#ArcOffBeforeMoveStd, WDAT2, WP4)
  LIN XP4
  ArcMainNG(#ArcOffAfterMoveStd, WDAT2, WP4)
;ENDFOLD
   $VEL.CP = 0.080
   LIN  {X -8.829, Y -5.312, Z 19.700, A 0.000, B 0.000, C 0.000} C_DIS

;FOLD ARCON WDAT1 LIN P3 Vel=0.5 m/s CPDAT1 Tool[1]:cmttorch Base[1]:vrashatel ;%{PE}
  ;FOLD Parameters ;%{h}
    ;Params IlfProvider=kukaroboter.arctech.arconlin; Kuka.IsGlobalPoint=False; Kuka.PointName=P3; Kuka.BlendingEnabled=False; Kuka.MoveDataName=CPDAT1; Kuka.VelocityPath=0.5; Kuka.CurrentCDSetIndex=0; Kuka.MovementParameterFieldEnabled=True; ArcTech.WdatVarName=WDAT1; ArcTech.Basic=3.4.3.1264
  ;ENDFOLD
  $BWDSTART = FALSE
  LDAT_ACT = LCPDAT1
  FDAT_ACT = FP3
  BAS(#CP_PARAMS, 0.5)
  SET_CD_PARAMS (0)
  TRIGGER WHEN DISTANCE = 1 DELAY = ArcGetDelay(#PreDefinition, WDAT1) DO ArcMainNG(#PreDefinition, WDAT1, WP3) PRIO = -1
  TRIGGER WHEN PATH = ArcGetPath(#OnTheFlyArcOn, WDAT1) DELAY = ArcGetDelay(#GasPreflow, WDAT1) DO ArcMainNG(#GasPreflow, WDAT1, WP3) PRIO = -1
  TRIGGER WHEN PATH = ArcGetPath(#OnTheFlyArcOn, WDAT1) DELAY = 0 DO ArcMainNG(#ArcOnMoveStd, WDAT1, WP3) PRIO = -1
  ArcMainNG(#ArcOnBeforeMoveStd, WDAT1, WP3)
  LIN XP3
  ArcMainNG(#ArcOnAfterMoveStd, WDAT1, WP3)
;ENDFOLD
   $VEL.CP = 0.060
   LIN  {X -5.312, Y -8.829, Z 19.700, A 0.000, B 0.000, C 0.000} C_DIS

;FOLD ARCOFF WDAT2 LIN P4 CPDAT2 Tool[1]:cmttorch Base[1]:vrashatel ;%{PE}
  ;FOLD Parameters ;%{h}
    ;Params IlfProvider=kukaroboter.arctech.arcofflin; Kuka.IsGlobalPoint=False; Kuka.PointName=P4; Kuka.BlendingEnabled=False; Kuka.MoveDataName=CPDAT2; Kuka.VelocityPath=0.01; Kuka.CurrentCDSetIndex=0; Kuka.MovementParameterFieldEnabled=True; ArcTech.WdatVarName=WDAT2; ArcTech.Basic=3.4.3.1264
  ;ENDFOLD
  $BWDSTART = FALSE
  LDAT_ACT = LCPDAT2
  FDAT_ACT = FP4
  BAS(#CP_PARAMS, gArcBasVelDefinition)
  SET_CD_PARAMS (0)
  TRIGGER WHEN PATH = ArcGetPath(#ArcOffBefore, WDAT2) DELAY = 0 DO ArcMainNG(#ArcOffBeforeOffStd, WDAT2, WP4) PRIO = -1
  TRIGGER WHEN PATH = ArcGetPath(#OnTheFlyArcOff, WDAT2) DELAY = 0 DO ArcMainNG(#ArcOffMoveStd, WDAT2, WP4) PRIO = -1
  ArcMainNG(#ArcOffBeforeMoveStd, WDAT2, WP4)
  LIN XP4
  ArcMainNG(#ArcOffAfterMoveStd, WDAT2, WP4)
;ENDFOLD
   $VEL.CP = 0.080
   LIN  {X -5.878, Y -8.829, Z 19.700, A 0.000, B 0.000, C 0.000} C_DIS

;FOLD ARCON WDAT1 LIN P3 Vel=0.5 m/s CPDAT1 Tool[1]:cmttorch Base[1]:vrashatel ;%{PE}
  ;FOLD Parameters ;%{h}
    ;Params IlfProvider=kukaroboter.arctech.arconlin; Kuka.IsGlobalPoint=False; Kuka.PointName=P3; Kuka.BlendingEnabled=False; Kuka.MoveDataName=CPDAT1; Kuka.VelocityPath=0.5; Kuka.CurrentCDSetIndex=0; Kuka.MovementParameterFieldEnabled=True; ArcTech.WdatVarName=WDAT1; ArcTech.Basic=3.4.3.1264
  ;ENDFOLD
  $BWDSTART = FALSE
  LDAT_ACT = LCPDAT1
  FDAT_ACT = FP3
  BAS(#CP_PARAMS, 0.5)
  SET_CD_PARAMS (0)
  TRIGGER WHEN DISTANCE = 1 DELAY = ArcGetDelay(#PreDefinition, WDAT1) DO ArcMainNG(#PreDefinition, WDAT1, WP3) PRIO = -1
  TRIGGER WHEN PATH = ArcGetPath(#OnTheFlyArcOn, WDAT1) DELAY = ArcGetDelay(#GasPreflow, WDAT1) DO ArcMainNG(#GasPreflow, WDAT1, WP3) PRIO = -1
  TRIGGER WHEN PATH = ArcGetPath(#OnTheFlyArcOn, WDAT1) DELAY = 0 DO ArcMainNG(#ArcOnMoveStd, WDAT1, WP3) PRIO = -1
  ArcMainNG(#ArcOnBeforeMoveStd, WDAT1, WP3)
  LIN XP3
  ArcMainNG(#ArcOnAfterMoveStd, WDAT1, WP3)
;ENDFOLD
   $VEL.CP = 0.060
   LIN  {X -8.829, Y -5.878, Z 19.700, A 0.000, B 0.000, C 0.000} C_DIS

;FOLD ARCOFF WDAT2 LIN P4 CPDAT2 Tool[1]:cmttorch Base[1]:vrashatel ;%{PE}
  ;FOLD Parameters ;%{h}
    ;Params IlfProvider=kukaroboter.arctech.arcofflin; Kuka.IsGlobalPoint=False; Kuka.PointName=P4; Kuka.BlendingEnabled=False; Kuka.MoveDataName=CPDAT2; Kuka.VelocityPath=0.01; Kuka.CurrentCDSetIndex=0; Kuka.MovementParameterFieldEnabled=True; ArcTech.WdatVarName=WDAT2; ArcTech.Basic=3.4.3.1264
  ;ENDFOLD
  $BWDSTART = FALSE
  LDAT_ACT = LCPDAT2
  FDAT_ACT = FP4
  BAS(#CP_PARAMS, gArcBasVelDefinition)
  SET_CD_PARAMS (0)
  TRIGGER WHEN PATH = ArcGetPath(#ArcOffBefore, WDAT2) DELAY = 0 DO ArcMainNG(#ArcOffBeforeOffStd, WDAT2, WP4) PRIO = -1
  TRIGGER WHEN PATH = ArcGetPath(#OnTheFlyArcOff, WDAT2) DELAY = 0 DO ArcMainNG(#ArcOffMoveStd, WDAT2, WP4) PRIO = -1
  ArcMainNG(#ArcOffBeforeMoveStd, WDAT2, WP4)
  LIN XP4
  ArcMainNG(#ArcOffAfterMoveStd, WDAT2, WP4)
;ENDFOLD
   $VEL.CP = 0.080
   LIN  {X -8.829, Y -6.443, Z 19.700, A 0.000, B 0.000, C 0.000} C_DIS

;FOLD ARCON WDAT1 LIN P3 Vel=0.5 m/s CPDAT1 Tool[1]:cmttorch Base[1]:vrashatel ;%{PE}
  ;FOLD Parameters ;%{h}
    ;Params IlfProvider=kukaroboter.arctech.arconlin; Kuka.IsGlobalPoint=False; Kuka.PointName=P3; Kuka.BlendingEnabled=False; Kuka.MoveDataName=CPDAT1; Kuka.VelocityPath=0.5; Kuka.CurrentCDSetIndex=0; Kuka.MovementParameterFieldEnabled=True; ArcTech.WdatVarName=WDAT1; ArcTech.Basic=3.4.3.1264
  ;ENDFOLD
  $BWDSTART = FALSE
  LDAT_ACT = LCPDAT1
  FDAT_ACT = FP3
  BAS(#CP_PARAMS, 0.5)
  SET_CD_PARAMS (0)
  TRIGGER WHEN DISTANCE = 1 DELAY = ArcGetDelay(#PreDefinition, WDAT1) DO ArcMainNG(#PreDefinition, WDAT1, WP3) PRIO = -1
  TRIGGER WHEN PATH = ArcGetPath(#OnTheFlyArcOn, WDAT1) DELAY = ArcGetDelay(#GasPreflow, WDAT1) DO ArcMainNG(#GasPreflow, WDAT1, WP3) PRIO = -1
  TRIGGER WHEN PATH = ArcGetPath(#OnTheFlyArcOn, WDAT1) DELAY = 0 DO ArcMainNG(#ArcOnMoveStd, WDAT1, WP3) PRIO = -1
  ArcMainNG(#ArcOnBeforeMoveStd, WDAT1, WP3)
  LIN XP3
  ArcMainNG(#ArcOnAfterMoveStd, WDAT1, WP3)
;ENDFOLD
   $VEL.CP = 0.060
   LIN  {X -6.443, Y -8.829, Z 19.700, A 0.000, B 0.000, C 0.000} C_DIS

;FOLD ARCOFF WDAT2 LIN P4 CPDAT2 Tool[1]:cmttorch Base[1]:vrashatel ;%{PE}
  ;FOLD Parameters ;%{h}
    ;Params IlfProvider=kukaroboter.arctech.arcofflin; Kuka.IsGlobalPoint=False; Kuka.PointName=P4; Kuka.BlendingEnabled=False; Kuka.MoveDataName=CPDAT2; Kuka.VelocityPath=0.01; Kuka.CurrentCDSetIndex=0; Kuka.MovementParameterFieldEnabled=True; ArcTech.WdatVarName=WDAT2; ArcTech.Basic=3.4.3.1264
  ;ENDFOLD
  $BWDSTART = FALSE
  LDAT_ACT = LCPDAT2
  FDAT_ACT = FP4
  BAS(#CP_PARAMS, gArcBasVelDefinition)
  SET_CD_PARAMS (0)
  TRIGGER WHEN PATH = ArcGetPath(#ArcOffBefore, WDAT2) DELAY = 0 DO ArcMainNG(#ArcOffBeforeOffStd, WDAT2, WP4) PRIO = -1
  TRIGGER WHEN PATH = ArcGetPath(#OnTheFlyArcOff, WDAT2) DELAY = 0 DO ArcMainNG(#ArcOffMoveStd, WDAT2, WP4) PRIO = -1
  ArcMainNG(#ArcOffBeforeMoveStd, WDAT2, WP4)
  LIN XP4
  ArcMainNG(#ArcOffAfterMoveStd, WDAT2, WP4)
;ENDFOLD
   $VEL.CP = 0.080
   LIN  {X -7.009, Y -8.829, Z 19.700, A 0.000, B 0.000, C 0.000} C_DIS

;FOLD ARCON WDAT1 LIN P3 Vel=0.5 m/s CPDAT1 Tool[1]:cmttorch Base[1]:vrashatel ;%{PE}
  ;FOLD Parameters ;%{h}
    ;Params IlfProvider=kukaroboter.arctech.arconlin; Kuka.IsGlobalPoint=False; Kuka.PointName=P3; Kuka.BlendingEnabled=False; Kuka.MoveDataName=CPDAT1; Kuka.VelocityPath=0.5; Kuka.CurrentCDSetIndex=0; Kuka.MovementParameterFieldEnabled=True; ArcTech.WdatVarName=WDAT1; ArcTech.Basic=3.4.3.1264
  ;ENDFOLD
  $BWDSTART = FALSE
  LDAT_ACT = LCPDAT1
  FDAT_ACT = FP3
  BAS(#CP_PARAMS, 0.5)
  SET_CD_PARAMS (0)
  TRIGGER WHEN DISTANCE = 1 DELAY = ArcGetDelay(#PreDefinition, WDAT1) DO ArcMainNG(#PreDefinition, WDAT1, WP3) PRIO = -1
  TRIGGER WHEN PATH = ArcGetPath(#OnTheFlyArcOn, WDAT1) DELAY = ArcGetDelay(#GasPreflow, WDAT1) DO ArcMainNG(#GasPreflow, WDAT1, WP3) PRIO = -1
  TRIGGER WHEN PATH = ArcGetPath(#OnTheFlyArcOn, WDAT1) DELAY = 0 DO ArcMainNG(#ArcOnMoveStd, WDAT1, WP3) PRIO = -1
  ArcMainNG(#ArcOnBeforeMoveStd, WDAT1, WP3)
  LIN XP3
  ArcMainNG(#ArcOnAfterMoveStd, WDAT1, WP3)
;ENDFOLD
   $VEL.CP = 0.060
   LIN  {X -8.829, Y -7.009, Z 19.700, A 0.000, B 0.000, C 0.000} C_DIS

;FOLD ARCOFF WDAT2 LIN P4 CPDAT2 Tool[1]:cmttorch Base[1]:vrashatel ;%{PE}
  ;FOLD Parameters ;%{h}
    ;Params IlfProvider=kukaroboter.arctech.arcofflin; Kuka.IsGlobalPoint=False; Kuka.PointName=P4; Kuka.BlendingEnabled=False; Kuka.MoveDataName=CPDAT2; Kuka.VelocityPath=0.01; Kuka.CurrentCDSetIndex=0; Kuka.MovementParameterFieldEnabled=True; ArcTech.WdatVarName=WDAT2; ArcTech.Basic=3.4.3.1264
  ;ENDFOLD
  $BWDSTART = FALSE
  LDAT_ACT = LCPDAT2
  FDAT_ACT = FP4
  BAS(#CP_PARAMS, gArcBasVelDefinition)
  SET_CD_PARAMS (0)
  TRIGGER WHEN PATH = ArcGetPath(#ArcOffBefore, WDAT2) DELAY = 0 DO ArcMainNG(#ArcOffBeforeOffStd, WDAT2, WP4) PRIO = -1
  TRIGGER WHEN PATH = ArcGetPath(#OnTheFlyArcOff, WDAT2) DELAY = 0 DO ArcMainNG(#ArcOffMoveStd, WDAT2, WP4) PRIO = -1
  ArcMainNG(#ArcOffBeforeMoveStd, WDAT2, WP4)
  LIN XP4
  ArcMainNG(#ArcOffAfterMoveStd, WDAT2, WP4)
;ENDFOLD
   $VEL.CP = 0.080
   LIN  {X -8.829, Y -7.575, Z 19.700, A 0.000, B 0.000, C 0.000} C_DIS

;FOLD ARCON WDAT1 LIN P3 Vel=0.5 m/s CPDAT1 Tool[1]:cmttorch Base[1]:vrashatel ;%{PE}
  ;FOLD Parameters ;%{h}
    ;Params IlfProvider=kukaroboter.arctech.arconlin; Kuka.IsGlobalPoint=False; Kuka.PointName=P3; Kuka.BlendingEnabled=False; Kuka.MoveDataName=CPDAT1; Kuka.VelocityPath=0.5; Kuka.CurrentCDSetIndex=0; Kuka.MovementParameterFieldEnabled=True; ArcTech.WdatVarName=WDAT1; ArcTech.Basic=3.4.3.1264
  ;ENDFOLD
  $BWDSTART = FALSE
  LDAT_ACT = LCPDAT1
  FDAT_ACT = FP3
  BAS(#CP_PARAMS, 0.5)
  SET_CD_PARAMS (0)
  TRIGGER WHEN DISTANCE = 1 DELAY = ArcGetDelay(#PreDefinition, WDAT1) DO ArcMainNG(#PreDefinition, WDAT1, WP3) PRIO = -1
  TRIGGER WHEN PATH = ArcGetPath(#OnTheFlyArcOn, WDAT1) DELAY = ArcGetDelay(#GasPreflow, WDAT1) DO ArcMainNG(#GasPreflow, WDAT1, WP3) PRIO = -1
  TRIGGER WHEN PATH = ArcGetPath(#OnTheFlyArcOn, WDAT1) DELAY = 0 DO ArcMainNG(#ArcOnMoveStd, WDAT1, WP3) PRIO = -1
  ArcMainNG(#ArcOnBeforeMoveStd, WDAT1, WP3)
  LIN XP3
  ArcMainNG(#ArcOnAfterMoveStd, WDAT1, WP3)
;ENDFOLD
   $VEL.CP = 0.060
   LIN  {X -7.575, Y -8.829, Z 19.700, A 0.000, B 0.000, C 0.000} C_DIS

;FOLD ARCOFF WDAT2 LIN P4 CPDAT2 Tool[1]:cmttorch Base[1]:vrashatel ;%{PE}
  ;FOLD Parameters ;%{h}
    ;Params IlfProvider=kukaroboter.arctech.arcofflin; Kuka.IsGlobalPoint=False; Kuka.PointName=P4; Kuka.BlendingEnabled=False; Kuka.MoveDataName=CPDAT2; Kuka.VelocityPath=0.01; Kuka.CurrentCDSetIndex=0; Kuka.MovementParameterFieldEnabled=True; ArcTech.WdatVarName=WDAT2; ArcTech.Basic=3.4.3.1264
  ;ENDFOLD
  $BWDSTART = FALSE
  LDAT_ACT = LCPDAT2
  FDAT_ACT = FP4
  BAS(#CP_PARAMS, gArcBasVelDefinition)
  SET_CD_PARAMS (0)
  TRIGGER WHEN PATH = ArcGetPath(#ArcOffBefore, WDAT2) DELAY = 0 DO ArcMainNG(#ArcOffBeforeOffStd, WDAT2, WP4) PRIO = -1
  TRIGGER WHEN PATH = ArcGetPath(#OnTheFlyArcOff, WDAT2) DELAY = 0 DO ArcMainNG(#ArcOffMoveStd, WDAT2, WP4) PRIO = -1
  ArcMainNG(#ArcOffBeforeMoveStd, WDAT2, WP4)
  LIN XP4
  ArcMainNG(#ArcOffAfterMoveStd, WDAT2, WP4)
;ENDFOLD
   $VEL.CP = 0.080
   LIN  {X -8.140, Y -8.829, Z 19.700, A 0.000, B 0.000, C 0.000} C_DIS

;FOLD ARCON WDAT1 LIN P3 Vel=0.5 m/s CPDAT1 Tool[1]:cmttorch Base[1]:vrashatel ;%{PE}
  ;FOLD Parameters ;%{h}
    ;Params IlfProvider=kukaroboter.arctech.arconlin; Kuka.IsGlobalPoint=False; Kuka.PointName=P3; Kuka.BlendingEnabled=False; Kuka.MoveDataName=CPDAT1; Kuka.VelocityPath=0.5; Kuka.CurrentCDSetIndex=0; Kuka.MovementParameterFieldEnabled=True; ArcTech.WdatVarName=WDAT1; ArcTech.Basic=3.4.3.1264
  ;ENDFOLD
  $BWDSTART = FALSE
  LDAT_ACT = LCPDAT1
  FDAT_ACT = FP3
  BAS(#CP_PARAMS, 0.5)
  SET_CD_PARAMS (0)
  TRIGGER WHEN DISTANCE = 1 DELAY = ArcGetDelay(#PreDefinition, WDAT1) DO ArcMainNG(#PreDefinition, WDAT1, WP3) PRIO = -1
  TRIGGER WHEN PATH = ArcGetPath(#OnTheFlyArcOn, WDAT1) DELAY = ArcGetDelay(#GasPreflow, WDAT1) DO ArcMainNG(#GasPreflow, WDAT1, WP3) PRIO = -1
  TRIGGER WHEN PATH = ArcGetPath(#OnTheFlyArcOn, WDAT1) DELAY = 0 DO ArcMainNG(#ArcOnMoveStd, WDAT1, WP3) PRIO = -1
  ArcMainNG(#ArcOnBeforeMoveStd, WDAT1, WP3)
  LIN XP3
  ArcMainNG(#ArcOnAfterMoveStd, WDAT1, WP3)
;ENDFOLD
   $VEL.CP = 0.060
   LIN  {X -8.829, Y -8.140, Z 19.700, A 0.000, B 0.000, C 0.000} C_DIS

;FOLD ARCOFF WDAT2 LIN P4 CPDAT2 Tool[1]:cmttorch Base[1]:vrashatel ;%{PE}
  ;FOLD Parameters ;%{h}
    ;Params IlfProvider=kukaroboter.arctech.arcofflin; Kuka.IsGlobalPoint=False; Kuka.PointName=P4; Kuka.BlendingEnabled=False; Kuka.MoveDataName=CPDAT2; Kuka.VelocityPath=0.01; Kuka.CurrentCDSetIndex=0; Kuka.MovementParameterFieldEnabled=True; ArcTech.WdatVarName=WDAT2; ArcTech.Basic=3.4.3.1264
  ;ENDFOLD
  $BWDSTART = FALSE
  LDAT_ACT = LCPDAT2
  FDAT_ACT = FP4
  BAS(#CP_PARAMS, gArcBasVelDefinition)
  SET_CD_PARAMS (0)
  TRIGGER WHEN PATH = ArcGetPath(#ArcOffBefore, WDAT2) DELAY = 0 DO ArcMainNG(#ArcOffBeforeOffStd, WDAT2, WP4) PRIO = -1
  TRIGGER WHEN PATH = ArcGetPath(#OnTheFlyArcOff, WDAT2) DELAY = 0 DO ArcMainNG(#ArcOffMoveStd, WDAT2, WP4) PRIO = -1
  ArcMainNG(#ArcOffBeforeMoveStd, WDAT2, WP4)
  LIN XP4
  ArcMainNG(#ArcOffAfterMoveStd, WDAT2, WP4)
;ENDFOLD
   $VEL.CP = 0.080
   LIN  {X -8.829, Y -8.706, Z 19.700, A 0.000, B 0.000, C 0.000} C_DIS

;FOLD ARCON WDAT1 LIN P3 Vel=0.5 m/s CPDAT1 Tool[1]:cmttorch Base[1]:vrashatel ;%{PE}
  ;FOLD Parameters ;%{h}
    ;Params IlfProvider=kukaroboter.arctech.arconlin; Kuka.IsGlobalPoint=False; Kuka.PointName=P3; Kuka.BlendingEnabled=False; Kuka.MoveDataName=CPDAT1; Kuka.VelocityPath=0.5; Kuka.CurrentCDSetIndex=0; Kuka.MovementParameterFieldEnabled=True; ArcTech.WdatVarName=WDAT1; ArcTech.Basic=3.4.3.1264
  ;ENDFOLD
  $BWDSTART = FALSE
  LDAT_ACT = LCPDAT1
  FDAT_ACT = FP3
  BAS(#CP_PARAMS, 0.5)
  SET_CD_PARAMS (0)
  TRIGGER WHEN DISTANCE = 1 DELAY = ArcGetDelay(#PreDefinition, WDAT1) DO ArcMainNG(#PreDefinition, WDAT1, WP3) PRIO = -1
  TRIGGER WHEN PATH = ArcGetPath(#OnTheFlyArcOn, WDAT1) DELAY = ArcGetDelay(#GasPreflow, WDAT1) DO ArcMainNG(#GasPreflow, WDAT1, WP3) PRIO = -1
  TRIGGER WHEN PATH = ArcGetPath(#OnTheFlyArcOn, WDAT1) DELAY = 0 DO ArcMainNG(#ArcOnMoveStd, WDAT1, WP3) PRIO = -1
  ArcMainNG(#ArcOnBeforeMoveStd, WDAT1, WP3)
  LIN XP3
  ArcMainNG(#ArcOnAfterMoveStd, WDAT1, WP3)
;ENDFOLD
   $VEL.CP = 0.060
   LIN  {X -8.706, Y -8.829, Z 19.700, A 0.000, B 0.000, C 0.000} C_DIS

;FOLD ARCOFF WDAT2 LIN P4 CPDAT2 Tool[1]:cmttorch Base[1]:vrashatel ;%{PE}
  ;FOLD Parameters ;%{h}
    ;Params IlfProvider=kukaroboter.arctech.arcofflin; Kuka.IsGlobalPoint=False; Kuka.PointName=P4; Kuka.BlendingEnabled=False; Kuka.MoveDataName=CPDAT2; Kuka.VelocityPath=0.01; Kuka.CurrentCDSetIndex=0; Kuka.MovementParameterFieldEnabled=True; ArcTech.WdatVarName=WDAT2; ArcTech.Basic=3.4.3.1264
  ;ENDFOLD
  $BWDSTART = FALSE
  LDAT_ACT = LCPDAT2
  FDAT_ACT = FP4
  BAS(#CP_PARAMS, gArcBasVelDefinition)
  SET_CD_PARAMS (0)
  TRIGGER WHEN PATH = ArcGetPath(#ArcOffBefore, WDAT2) DELAY = 0 DO ArcMainNG(#ArcOffBeforeOffStd, WDAT2, WP4) PRIO = -1
  TRIGGER WHEN PATH = ArcGetPath(#OnTheFlyArcOff, WDAT2) DELAY = 0 DO ArcMainNG(#ArcOffMoveStd, WDAT2, WP4) PRIO = -1
  ArcMainNG(#ArcOffBeforeMoveStd, WDAT2, WP4)
  LIN XP4
  ArcMainNG(#ArcOffAfterMoveStd, WDAT2, WP4)
;ENDFOLD
   $VEL.CP = 0.080
   LIN  {X -8.706, Y -9.200, Z 19.700, A 0.000, B 0.000, C 0.000} C_DIS
   $VEL.CP = 0.010
   LIN  {X -8.706, Y -9.200, Z 19.900, A 0.000, B 0.000, C 0.000} C_DIS
   $VEL.CP = 0.080
   LIN  {X -8.706, Y -9.290, Z 19.900, A 0.000, B 0.000, C 0.000} C_DIS
   $VEL.CP = 0.080
   LIN  {X -9.218, Y -9.218, Z 19.900, A 0.000, B 0.000, C 0.000} C_DIS
   $VEL.CP = 0.080
   LIN  {X -9.530, Y 9.530, Z 19.900, A 0.000, B 0.000, C 0.000} C_DIS
   $VEL.CP = 0.080
   LIN  {X -9.800, Y 9.800, Z 19.900, A 0.000, B 0.000, C 0.000} C_DIS

;FOLD ARCON WDAT1 LIN P3 Vel=0.5 m/s CPDAT1 Tool[1]:cmttorch Base[1]:vrashatel ;%{PE}
  ;FOLD Parameters ;%{h}
    ;Params IlfProvider=kukaroboter.arctech.arconlin; Kuka.IsGlobalPoint=False; Kuka.PointName=P3; Kuka.BlendingEnabled=False; Kuka.MoveDataName=CPDAT1; Kuka.VelocityPath=0.5; Kuka.CurrentCDSetIndex=0; Kuka.MovementParameterFieldEnabled=True; ArcTech.WdatVarName=WDAT1; ArcTech.Basic=3.4.3.1264
  ;ENDFOLD
  $BWDSTART = FALSE
  LDAT_ACT = LCPDAT1
  FDAT_ACT = FP3
  BAS(#CP_PARAMS, 0.5)
  SET_CD_PARAMS (0)
  TRIGGER WHEN DISTANCE = 1 DELAY = ArcGetDelay(#PreDefinition, WDAT1) DO ArcMainNG(#PreDefinition, WDAT1, WP3) PRIO = -1
  TRIGGER WHEN PATH = ArcGetPath(#OnTheFlyArcOn, WDAT1) DELAY = ArcGetDelay(#GasPreflow, WDAT1) DO ArcMainNG(#GasPreflow, WDAT1, WP3) PRIO = -1
  TRIGGER WHEN PATH = ArcGetPath(#OnTheFlyArcOn, WDAT1) DELAY = 0 DO ArcMainNG(#ArcOnMoveStd, WDAT1, WP3) PRIO = -1
  ArcMainNG(#ArcOnBeforeMoveStd, WDAT1, WP3)
  LIN XP3
  ArcMainNG(#ArcOnAfterMoveStd, WDAT1, WP3)
;ENDFOLD
   $VEL.CP = 0.025
   LIN  {X -9.800, Y 9.800, Z 19.900, A 0.000, B 0.000, C 0.000} C_DIS
   $VEL.CP = 0.060
   LIN  {X -9.800, Y -9.800, Z 19.900, A 0.000, B 0.000, C 0.000} C_DIS
   $VEL.CP = 0.060
   LIN  {X 9.800, Y -9.800, Z 19.900, A 0.000, B 0.000, C 0.000} C_DIS
   $VEL.CP = 0.060
   LIN  {X 9.800, Y 9.800, Z 19.900, A 0.000, B 0.000, C 0.000} C_DIS
   $VEL.CP = 0.060
   LIN  {X -9.800, Y 9.800, Z 19.900, A 0.000, B 0.000, C 0.000} C_DIS

;FOLD ARCOFF WDAT2 LIN P4 CPDAT2 Tool[1]:cmttorch Base[1]:vrashatel ;%{PE}
  ;FOLD Parameters ;%{h}
    ;Params IlfProvider=kukaroboter.arctech.arcofflin; Kuka.IsGlobalPoint=False; Kuka.PointName=P4; Kuka.BlendingEnabled=False; Kuka.MoveDataName=CPDAT2; Kuka.VelocityPath=0.01; Kuka.CurrentCDSetIndex=0; Kuka.MovementParameterFieldEnabled=True; ArcTech.WdatVarName=WDAT2; ArcTech.Basic=3.4.3.1264
  ;ENDFOLD
  $BWDSTART = FALSE
  LDAT_ACT = LCPDAT2
  FDAT_ACT = FP4
  BAS(#CP_PARAMS, gArcBasVelDefinition)
  SET_CD_PARAMS (0)
  TRIGGER WHEN PATH = ArcGetPath(#ArcOffBefore, WDAT2) DELAY = 0 DO ArcMainNG(#ArcOffBeforeOffStd, WDAT2, WP4) PRIO = -1
  TRIGGER WHEN PATH = ArcGetPath(#OnTheFlyArcOff, WDAT2) DELAY = 0 DO ArcMainNG(#ArcOffMoveStd, WDAT2, WP4) PRIO = -1
  ArcMainNG(#ArcOffBeforeMoveStd, WDAT2, WP4)
  LIN XP4
  ArcMainNG(#ArcOffAfterMoveStd, WDAT2, WP4)
;ENDFOLD
   $VEL.CP = 0.080
   LIN  {X -9.800, Y 9.600, Z 19.900, A 0.000, B 0.000, C 0.000} C_DIS
   $VEL.CP = 0.080
   LIN  {X -9.360, Y 9.360, Z 19.900, A 0.000, B 0.000, C 0.000} C_DIS
   $VEL.CP = 0.080
   LIN  {X -4.094, Y 9.190, Z 19.900, A 0.000, B 0.000, C 0.000} C_DIS
   $VEL.CP = 0.080
   LIN  {X -4.094, Y 7.108, Z 19.900, A 0.000, B 0.000, C 0.000} C_DIS
   $VEL.CP = 0.080
   LIN  {X -4.094, Y 4.605, Z 19.900, A 0.000, B 0.000, C 0.000} C_DIS
   $VEL.CP = 0.080
   LIN  {X -3.794, Y 4.605, Z 19.900, A 0.000, B 0.000, C 0.000} C_DIS

;FOLD ARCON WDAT1 LIN P3 Vel=0.5 m/s CPDAT1 Tool[1]:cmttorch Base[1]:vrashatel ;%{PE}
  ;FOLD Parameters ;%{h}
    ;Params IlfProvider=kukaroboter.arctech.arconlin; Kuka.IsGlobalPoint=False; Kuka.PointName=P3; Kuka.BlendingEnabled=False; Kuka.MoveDataName=CPDAT1; Kuka.VelocityPath=0.5; Kuka.CurrentCDSetIndex=0; Kuka.MovementParameterFieldEnabled=True; ArcTech.WdatVarName=WDAT1; ArcTech.Basic=3.4.3.1264
  ;ENDFOLD
  $BWDSTART = FALSE
  LDAT_ACT = LCPDAT1
  FDAT_ACT = FP3
  BAS(#CP_PARAMS, 0.5)
  SET_CD_PARAMS (0)
  TRIGGER WHEN DISTANCE = 1 DELAY = ArcGetDelay(#PreDefinition, WDAT1) DO ArcMainNG(#PreDefinition, WDAT1, WP3) PRIO = -1
  TRIGGER WHEN PATH = ArcGetPath(#OnTheFlyArcOn, WDAT1) DELAY = ArcGetDelay(#GasPreflow, WDAT1) DO ArcMainNG(#GasPreflow, WDAT1, WP3) PRIO = -1
  TRIGGER WHEN PATH = ArcGetPath(#OnTheFlyArcOn, WDAT1) DELAY = 0 DO ArcMainNG(#ArcOnMoveStd, WDAT1, WP3) PRIO = -1
  ArcMainNG(#ArcOnBeforeMoveStd, WDAT1, WP3)
  LIN XP3
  ArcMainNG(#ArcOnAfterMoveStd, WDAT1, WP3)
;ENDFOLD
   $VEL.CP = 0.025
   LIN  {X -3.794, Y 4.605, Z 19.900, A 0.000, B 0.000, C 0.000} C_DIS
   $VEL.CP = 0.060
   LIN  {X -3.794, Y 6.518, Z 19.900, A 0.000, B 0.000, C 0.000} C_DIS
   $VEL.CP = 0.060
   LIN  {X 4.127, Y 6.518, Z 19.900, A 0.000, B 0.000, C 0.000} C_DIS
   $VEL.CP = 0.060
   LIN  {X 4.127, Y 5.892, Z 19.900, A 0.000, B 0.000, C 0.000} C_DIS
   $VEL.CP = 0.060
   LIN  {X -1.058, Y -4.280, Z 19.900, A 0.000, B 0.000, C 0.000} C_DIS
   $VEL.CP = 0.060
   LIN  {X 4.312, Y -4.280, Z 19.900, A 0.000, B 0.000, C 0.000} C_DIS
   $VEL.CP = 0.060
   LIN  {X 4.312, Y -6.193, Z 19.900, A 0.000, B 0.000, C 0.000} C_DIS
   $VEL.CP = 0.060
   LIN  {X -3.878, Y -6.193, Z 19.900, A 0.000, B 0.000, C 0.000} C_DIS
   $VEL.CP = 0.060
   LIN  {X -3.878, Y -5.567, Z 19.900, A 0.000, B 0.000, C 0.000} C_DIS
   $VEL.CP = 0.060
   LIN  {X 1.290, Y 4.605, Z 19.900, A 0.000, B 0.000, C 0.000} C_DIS
   $VEL.CP = 0.060
   LIN  {X -3.794, Y 4.605, Z 19.900, A 0.000, B 0.000, C 0.000} C_DIS

;FOLD ARCOFF WDAT2 LIN P4 CPDAT2 Tool[1]:cmttorch Base[1]:vrashatel ;%{PE}
  ;FOLD Parameters ;%{h}
    ;Params IlfProvider=kukaroboter.arctech.arcofflin; Kuka.IsGlobalPoint=False; Kuka.PointName=P4; Kuka.BlendingEnabled=False; Kuka.MoveDataName=CPDAT2; Kuka.VelocityPath=0.01; Kuka.CurrentCDSetIndex=0; Kuka.MovementParameterFieldEnabled=True; ArcTech.WdatVarName=WDAT2; ArcTech.Basic=3.4.3.1264
  ;ENDFOLD
  $BWDSTART = FALSE
  LDAT_ACT = LCPDAT2
  FDAT_ACT = FP4
  BAS(#CP_PARAMS, gArcBasVelDefinition)
  SET_CD_PARAMS (0)
  TRIGGER WHEN PATH = ArcGetPath(#ArcOffBefore, WDAT2) DELAY = 0 DO ArcMainNG(#ArcOffBeforeOffStd, WDAT2, WP4) PRIO = -1
  TRIGGER WHEN PATH = ArcGetPath(#OnTheFlyArcOff, WDAT2) DELAY = 0 DO ArcMainNG(#ArcOffMoveStd, WDAT2, WP4) PRIO = -1
  ArcMainNG(#ArcOffBeforeMoveStd, WDAT2, WP4)
  LIN XP4
  ArcMainNG(#ArcOffAfterMoveStd, WDAT2, WP4)
;ENDFOLD
   $VEL.CP = 0.080
   LIN  {X -3.794, Y 4.805, Z 19.900, A 0.000, B 0.000, C 0.000} C_DIS
   $VEL.CP = 0.080
   LIN  {X -4.194, Y 4.205, Z 19.900, A 0.000, B 0.000, C 0.000} C_DIS

;FOLD ARCON WDAT1 LIN P3 Vel=0.5 m/s CPDAT1 Tool[1]:cmttorch Base[1]:vrashatel ;%{PE}
  ;FOLD Parameters ;%{h}
    ;Params IlfProvider=kukaroboter.arctech.arconlin; Kuka.IsGlobalPoint=False; Kuka.PointName=P3; Kuka.BlendingEnabled=False; Kuka.MoveDataName=CPDAT1; Kuka.VelocityPath=0.5; Kuka.CurrentCDSetIndex=0; Kuka.MovementParameterFieldEnabled=True; ArcTech.WdatVarName=WDAT1; ArcTech.Basic=3.4.3.1264
  ;ENDFOLD
  $BWDSTART = FALSE
  LDAT_ACT = LCPDAT1
  FDAT_ACT = FP3
  BAS(#CP_PARAMS, 0.5)
  SET_CD_PARAMS (0)
  TRIGGER WHEN DISTANCE = 1 DELAY = ArcGetDelay(#PreDefinition, WDAT1) DO ArcMainNG(#PreDefinition, WDAT1, WP3) PRIO = -1
  TRIGGER WHEN PATH = ArcGetPath(#OnTheFlyArcOn, WDAT1) DELAY = ArcGetDelay(#GasPreflow, WDAT1) DO ArcMainNG(#GasPreflow, WDAT1, WP3) PRIO = -1
  TRIGGER WHEN PATH = ArcGetPath(#OnTheFlyArcOn, WDAT1) DELAY = 0 DO ArcMainNG(#ArcOnMoveStd, WDAT1, WP3) PRIO = -1
  ArcMainNG(#ArcOnBeforeMoveStd, WDAT1, WP3)
  LIN XP3
  ArcMainNG(#ArcOnAfterMoveStd, WDAT1, WP3)
;ENDFOLD
   $VEL.CP = 0.060
   LIN  {X -4.194, Y 6.918, Z 19.900, A 0.000, B 0.000, C 0.000} C_DIS
   $VEL.CP = 0.060
   LIN  {X 4.527, Y 6.918, Z 19.900, A 0.000, B 0.000, C 0.000} C_DIS
   $VEL.CP = 0.060
   LIN  {X 4.527, Y 5.796, Z 19.900, A 0.000, B 0.000, C 0.000} C_DIS
   $VEL.CP = 0.060
   LIN  {X -0.405, Y -3.880, Z 19.900, A 0.000, B 0.000, C 0.000} C_DIS
   $VEL.CP = 0.060
   LIN  {X 4.712, Y -3.880, Z 19.900, A 0.000, B 0.000, C 0.000} C_DIS
   $VEL.CP = 0.060
   LIN  {X 4.712, Y -6.593, Z 19.900, A 0.000, B 0.000, C 0.000} C_DIS
   $VEL.CP = 0.060
   LIN  {X -4.278, Y -6.593, Z 19.900, A 0.000, B 0.000, C 0.000} C_DIS
   $VEL.CP = 0.060
   LIN  {X -4.278, Y -5.471, Z 19.900, A 0.000, B 0.000, C 0.000} C_DIS
   $VEL.CP = 0.060
   LIN  {X 0.638, Y 4.205, Z 19.900, A 0.000, B 0.000, C 0.000} C_DIS
   $VEL.CP = 0.060
   LIN  {X -4.194, Y 4.205, Z 19.900, A 0.000, B 0.000, C 0.000} C_DIS

;FOLD ARCOFF WDAT2 LIN P4 CPDAT2 Tool[1]:cmttorch Base[1]:vrashatel ;%{PE}
  ;FOLD Parameters ;%{h}
    ;Params IlfProvider=kukaroboter.arctech.arcofflin; Kuka.IsGlobalPoint=False; Kuka.PointName=P4; Kuka.BlendingEnabled=False; Kuka.MoveDataName=CPDAT2; Kuka.VelocityPath=0.01; Kuka.CurrentCDSetIndex=0; Kuka.MovementParameterFieldEnabled=True; ArcTech.WdatVarName=WDAT2; ArcTech.Basic=3.4.3.1264
  ;ENDFOLD
  $BWDSTART = FALSE
  LDAT_ACT = LCPDAT2
  FDAT_ACT = FP4
  BAS(#CP_PARAMS, gArcBasVelDefinition)
  SET_CD_PARAMS (0)
  TRIGGER WHEN PATH = ArcGetPath(#ArcOffBefore, WDAT2) DELAY = 0 DO ArcMainNG(#ArcOffBeforeOffStd, WDAT2, WP4) PRIO = -1
  TRIGGER WHEN PATH = ArcGetPath(#OnTheFlyArcOff, WDAT2) DELAY = 0 DO ArcMainNG(#ArcOffMoveStd, WDAT2, WP4) PRIO = -1
  ArcMainNG(#ArcOffBeforeMoveStd, WDAT2, WP4)
  LIN XP4
  ArcMainNG(#ArcOffAfterMoveStd, WDAT2, WP4)
;ENDFOLD
   $VEL.CP = 0.080
   LIN  {X -4.390, Y 7.114, Z 19.900, A 0.000, B 0.000, C 0.000} C_DIS
   $VEL.CP = 0.080
   LIN  {X -4.390, Y 9.190, Z 19.900, A 0.000, B 0.000, C 0.000} C_DIS
   $VEL.CP = 0.080
   LIN  {X -9.400, Y 9.400, Z 19.900, A 0.000, B 0.000, C 0.000} C_DIS

;FOLD ARCON WDAT1 LIN P3 Vel=0.5 m/s CPDAT1 Tool[1]:cmttorch Base[1]:vrashatel ;%{PE}
  ;FOLD Parameters ;%{h}
    ;Params IlfProvider=kukaroboter.arctech.arconlin; Kuka.IsGlobalPoint=False; Kuka.PointName=P3; Kuka.BlendingEnabled=False; Kuka.MoveDataName=CPDAT1; Kuka.VelocityPath=0.5; Kuka.CurrentCDSetIndex=0; Kuka.MovementParameterFieldEnabled=True; ArcTech.WdatVarName=WDAT1; ArcTech.Basic=3.4.3.1264
  ;ENDFOLD
  $BWDSTART = FALSE
  LDAT_ACT = LCPDAT1
  FDAT_ACT = FP3
  BAS(#CP_PARAMS, 0.5)
  SET_CD_PARAMS (0)
  TRIGGER WHEN DISTANCE = 1 DELAY = ArcGetDelay(#PreDefinition, WDAT1) DO ArcMainNG(#PreDefinition, WDAT1, WP3) PRIO = -1
  TRIGGER WHEN PATH = ArcGetPath(#OnTheFlyArcOn, WDAT1) DELAY = ArcGetDelay(#GasPreflow, WDAT1) DO ArcMainNG(#GasPreflow, WDAT1, WP3) PRIO = -1
  TRIGGER WHEN PATH = ArcGetPath(#OnTheFlyArcOn, WDAT1) DELAY = 0 DO ArcMainNG(#ArcOnMoveStd, WDAT1, WP3) PRIO = -1
  ArcMainNG(#ArcOnBeforeMoveStd, WDAT1, WP3)
  LIN XP3
  ArcMainNG(#ArcOnAfterMoveStd, WDAT1, WP3)
;ENDFOLD
   $VEL.CP = 0.025
   LIN  {X -9.400, Y 9.400, Z 19.900, A 0.000, B 0.000, C 0.000} C_DIS
   $VEL.CP = 0.060
   LIN  {X -9.400, Y -9.400, Z 19.900, A 0.000, B 0.000, C 0.000} C_DIS
   $VEL.CP = 0.060
   LIN  {X 9.400, Y -9.400, Z 19.900, A 0.000, B 0.000, C 0.000} C_DIS
   $VEL.CP = 0.060
   LIN  {X 9.400, Y 9.400, Z 19.900, A 0.000, B 0.000, C 0.000} C_DIS
   $VEL.CP = 0.060
   LIN  {X -9.400, Y 9.400, Z 19.900, A 0.000, B 0.000, C 0.000} C_DIS

;FOLD ARCOFF WDAT2 LIN P4 CPDAT2 Tool[1]:cmttorch Base[1]:vrashatel ;%{PE}
  ;FOLD Parameters ;%{h}
    ;Params IlfProvider=kukaroboter.arctech.arcofflin; Kuka.IsGlobalPoint=False; Kuka.PointName=P4; Kuka.BlendingEnabled=False; Kuka.MoveDataName=CPDAT2; Kuka.VelocityPath=0.01; Kuka.CurrentCDSetIndex=0; Kuka.MovementParameterFieldEnabled=True; ArcTech.WdatVarName=WDAT2; ArcTech.Basic=3.4.3.1264
  ;ENDFOLD
  $BWDSTART = FALSE
  LDAT_ACT = LCPDAT2
  FDAT_ACT = FP4
  BAS(#CP_PARAMS, gArcBasVelDefinition)
  SET_CD_PARAMS (0)
  TRIGGER WHEN PATH = ArcGetPath(#ArcOffBefore, WDAT2) DELAY = 0 DO ArcMainNG(#ArcOffBeforeOffStd, WDAT2, WP4) PRIO = -1
  TRIGGER WHEN PATH = ArcGetPath(#OnTheFlyArcOff, WDAT2) DELAY = 0 DO ArcMainNG(#ArcOffMoveStd, WDAT2, WP4) PRIO = -1
  ArcMainNG(#ArcOffBeforeMoveStd, WDAT2, WP4)
  LIN XP4
  ArcMainNG(#ArcOffAfterMoveStd, WDAT2, WP4)
;ENDFOLD
   $VEL.CP = 0.080
   LIN  {X -9.010, Y 9.010, Z 19.900, A 0.000, B 0.000, C 0.000} C_DIS

;FOLD ARCON WDAT1 LIN P3 Vel=0.5 m/s CPDAT1 Tool[1]:cmttorch Base[1]:vrashatel ;%{PE}
  ;FOLD Parameters ;%{h}
    ;Params IlfProvider=kukaroboter.arctech.arconlin; Kuka.IsGlobalPoint=False; Kuka.PointName=P3; Kuka.BlendingEnabled=False; Kuka.MoveDataName=CPDAT1; Kuka.VelocityPath=0.5; Kuka.CurrentCDSetIndex=0; Kuka.MovementParameterFieldEnabled=True; ArcTech.WdatVarName=WDAT1; ArcTech.Basic=3.4.3.1264
  ;ENDFOLD
  $BWDSTART = FALSE
  LDAT_ACT = LCPDAT1
  FDAT_ACT = FP3
  BAS(#CP_PARAMS, 0.5)
  SET_CD_PARAMS (0)
  TRIGGER WHEN DISTANCE = 1 DELAY = ArcGetDelay(#PreDefinition, WDAT1) DO ArcMainNG(#PreDefinition, WDAT1, WP3) PRIO = -1
  TRIGGER WHEN PATH = ArcGetPath(#OnTheFlyArcOn, WDAT1) DELAY = ArcGetDelay(#GasPreflow, WDAT1) DO ArcMainNG(#GasPreflow, WDAT1, WP3) PRIO = -1
  TRIGGER WHEN PATH = ArcGetPath(#OnTheFlyArcOn, WDAT1) DELAY = 0 DO ArcMainNG(#ArcOnMoveStd, WDAT1, WP3) PRIO = -1
  ArcMainNG(#ArcOnBeforeMoveStd, WDAT1, WP3)
  LIN XP3
  ArcMainNG(#ArcOnAfterMoveStd, WDAT1, WP3)
;ENDFOLD
   $VEL.CP = 0.060
   LIN  {X -9.010, Y -9.010, Z 19.900, A 0.000, B 0.000, C 0.000} C_DIS
   $VEL.CP = 0.060
   LIN  {X 9.010, Y -9.010, Z 19.900, A 0.000, B 0.000, C 0.000} C_DIS
   $VEL.CP = 0.060
   LIN  {X 9.010, Y 9.010, Z 19.900, A 0.000, B 0.000, C 0.000} C_DIS
   $VEL.CP = 0.060
   LIN  {X -9.010, Y 9.010, Z 19.900, A 0.000, B 0.000, C 0.000} C_DIS

;FOLD ARCOFF WDAT2 LIN P4 CPDAT2 Tool[1]:cmttorch Base[1]:vrashatel ;%{PE}
  ;FOLD Parameters ;%{h}
    ;Params IlfProvider=kukaroboter.arctech.arcofflin; Kuka.IsGlobalPoint=False; Kuka.PointName=P4; Kuka.BlendingEnabled=False; Kuka.MoveDataName=CPDAT2; Kuka.VelocityPath=0.01; Kuka.CurrentCDSetIndex=0; Kuka.MovementParameterFieldEnabled=True; ArcTech.WdatVarName=WDAT2; ArcTech.Basic=3.4.3.1264
  ;ENDFOLD
  $BWDSTART = FALSE
  LDAT_ACT = LCPDAT2
  FDAT_ACT = FP4
  BAS(#CP_PARAMS, gArcBasVelDefinition)
  SET_CD_PARAMS (0)
  TRIGGER WHEN PATH = ArcGetPath(#ArcOffBefore, WDAT2) DELAY = 0 DO ArcMainNG(#ArcOffBeforeOffStd, WDAT2, WP4) PRIO = -1
  TRIGGER WHEN PATH = ArcGetPath(#OnTheFlyArcOff, WDAT2) DELAY = 0 DO ArcMainNG(#ArcOffMoveStd, WDAT2, WP4) PRIO = -1
  ArcMainNG(#ArcOffBeforeMoveStd, WDAT2, WP4)
  LIN XP4
  ArcMainNG(#ArcOffAfterMoveStd, WDAT2, WP4)
;ENDFOLD
   $VEL.CP = 0.080
   LIN  {X -9.290, Y 9.010, Z 19.900, A 0.000, B 0.000, C 0.000} C_DIS
   $VEL.CP = 0.080
   LIN  {X -9.218, Y 9.218, Z 19.900, A 0.000, B 0.000, C 0.000} C_DIS
   $VEL.CP = 0.080
   LIN  {X -4.304, Y 9.190, Z 19.900, A 0.000, B 0.000, C 0.000} C_DIS
   $VEL.CP = 0.080
   LIN  {X -4.304, Y 7.108, Z 19.900, A 0.000, B 0.000, C 0.000} C_DIS
   $VEL.CP = 0.080
   LIN  {X -4.584, Y 7.308, Z 19.900, A 0.000, B 0.000, C 0.000} C_DIS

;FOLD ARCON WDAT1 LIN P3 Vel=0.5 m/s CPDAT1 Tool[1]:cmttorch Base[1]:vrashatel ;%{PE}
  ;FOLD Parameters ;%{h}
    ;Params IlfProvider=kukaroboter.arctech.arconlin; Kuka.IsGlobalPoint=False; Kuka.PointName=P3; Kuka.BlendingEnabled=False; Kuka.MoveDataName=CPDAT1; Kuka.VelocityPath=0.5; Kuka.CurrentCDSetIndex=0; Kuka.MovementParameterFieldEnabled=True; ArcTech.WdatVarName=WDAT1; ArcTech.Basic=3.4.3.1264
  ;ENDFOLD
  $BWDSTART = FALSE
  LDAT_ACT = LCPDAT1
  FDAT_ACT = FP3
  BAS(#CP_PARAMS, 0.5)
  SET_CD_PARAMS (0)
  TRIGGER WHEN DISTANCE = 1 DELAY = ArcGetDelay(#PreDefinition, WDAT1) DO ArcMainNG(#PreDefinition, WDAT1, WP3) PRIO = -1
  TRIGGER WHEN PATH = ArcGetPath(#OnTheFlyArcOn, WDAT1) DELAY = ArcGetDelay(#GasPreflow, WDAT1) DO ArcMainNG(#GasPreflow, WDAT1, WP3) PRIO = -1
  TRIGGER WHEN PATH = ArcGetPath(#OnTheFlyArcOn, WDAT1) DELAY = 0 DO ArcMainNG(#ArcOnMoveStd, WDAT1, WP3) PRIO = -1
  ArcMainNG(#ArcOnBeforeMoveStd, WDAT1, WP3)
  LIN XP3
  ArcMainNG(#ArcOnAfterMoveStd, WDAT1, WP3)
;ENDFOLD
   $VEL.CP = 0.025
   LIN  {X -4.584, Y 7.308, Z 19.900, A 0.000, B 0.000, C 0.000} C_DIS
   $VEL.CP = 0.060
   LIN  {X 4.917, Y 7.308, Z 19.900, A 0.000, B 0.000, C 0.000} C_DIS
   $VEL.CP = 0.060
   LIN  {X 4.917, Y 5.702, Z 19.900, A 0.000, B 0.000, C 0.000} C_DIS
   $VEL.CP = 0.060
   LIN  {X 0.231, Y -3.490, Z 19.900, A 0.000, B 0.000, C 0.000} C_DIS
   $VEL.CP = 0.060
   LIN  {X 5.102, Y -3.490, Z 19.900, A 0.000, B 0.000, C 0.000} C_DIS
   $VEL.CP = 0.060
   LIN  {X 5.102, Y -6.983, Z 19.900, A 0.000, B 0.000, C 0.000} C_DIS
   $VEL.CP = 0.060
   LIN  {X -4.668, Y -6.983, Z 19.900, A 0.000, B 0.000, C 0.000} C_DIS
   $VEL.CP = 0.060
   LIN  {X -4.668, Y -5.378, Z 19.900, A 0.000, B 0.000, C 0.000} C_DIS
   $VEL.CP = 0.060
   LIN  {X 0.003, Y 3.815, Z 19.900, A 0.000, B 0.000, C 0.000} C_DIS
   $VEL.CP = 0.060
   LIN  {X -4.584, Y 3.815, Z 19.900, A 0.000, B 0.000, C 0.000} C_DIS
   $VEL.CP = 0.060
   LIN  {X -4.584, Y 7.308, Z 19.900, A 0.000, B 0.000, C 0.000} C_DIS

;FOLD ARCOFF WDAT2 LIN P4 CPDAT2 Tool[1]:cmttorch Base[1]:vrashatel ;%{PE}
  ;FOLD Parameters ;%{h}
    ;Params IlfProvider=kukaroboter.arctech.arcofflin; Kuka.IsGlobalPoint=False; Kuka.PointName=P4; Kuka.BlendingEnabled=False; Kuka.MoveDataName=CPDAT2; Kuka.VelocityPath=0.01; Kuka.CurrentCDSetIndex=0; Kuka.MovementParameterFieldEnabled=True; ArcTech.WdatVarName=WDAT2; ArcTech.Basic=3.4.3.1264
  ;ENDFOLD
  $BWDSTART = FALSE
  LDAT_ACT = LCPDAT2
  FDAT_ACT = FP4
  BAS(#CP_PARAMS, gArcBasVelDefinition)
  SET_CD_PARAMS (0)
  TRIGGER WHEN PATH = ArcGetPath(#ArcOffBefore, WDAT2) DELAY = 0 DO ArcMainNG(#ArcOffBeforeOffStd, WDAT2, WP4) PRIO = -1
  TRIGGER WHEN PATH = ArcGetPath(#OnTheFlyArcOff, WDAT2) DELAY = 0 DO ArcMainNG(#ArcOffMoveStd, WDAT2, WP4) PRIO = -1
  ArcMainNG(#ArcOffBeforeMoveStd, WDAT2, WP4)
  LIN XP4
  ArcMainNG(#ArcOffAfterMoveStd, WDAT2, WP4)
;ENDFOLD
   $VEL.CP = 0.080
   LIN  {X -4.304, Y 7.058, Z 19.900, A 0.000, B 0.000, C 0.000} C_DIS
   $VEL.CP = 0.080
   LIN  {X -4.390, Y 7.114, Z 19.900, A 0.000, B 0.000, C 0.000} C_DIS
   $VEL.CP = 0.080
   LIN  {X -9.190, Y 7.114, Z 19.900, A 0.000, B 0.000, C 0.000} C_DIS
   $VEL.CP = 0.080
   LIN  {X -9.290, Y 8.706, Z 19.900, A 0.000, B 0.000, C 0.000} C_DIS
   $VEL.CP = 0.080
   LIN  {X -8.829, Y 8.706, Z 19.900, A 0.000, B 0.000, C 0.000} C_DIS

;FOLD ARCON WDAT1 LIN P3 Vel=0.5 m/s CPDAT1 Tool[1]:cmttorch Base[1]:vrashatel ;%{PE}
  ;FOLD Parameters ;%{h}
    ;Params IlfProvider=kukaroboter.arctech.arconlin; Kuka.IsGlobalPoint=False; Kuka.PointName=P3; Kuka.BlendingEnabled=False; Kuka.MoveDataName=CPDAT1; Kuka.VelocityPath=0.5; Kuka.CurrentCDSetIndex=0; Kuka.MovementParameterFieldEnabled=True; ArcTech.WdatVarName=WDAT1; ArcTech.Basic=3.4.3.1264
  ;ENDFOLD
  $BWDSTART = FALSE
  LDAT_ACT = LCPDAT1
  FDAT_ACT = FP3
  BAS(#CP_PARAMS, 0.5)
  SET_CD_PARAMS (0)
  TRIGGER WHEN DISTANCE = 1 DELAY = ArcGetDelay(#PreDefinition, WDAT1) DO ArcMainNG(#PreDefinition, WDAT1, WP3) PRIO = -1
  TRIGGER WHEN PATH = ArcGetPath(#OnTheFlyArcOn, WDAT1) DELAY = ArcGetDelay(#GasPreflow, WDAT1) DO ArcMainNG(#GasPreflow, WDAT1, WP3) PRIO = -1
  TRIGGER WHEN PATH = ArcGetPath(#OnTheFlyArcOn, WDAT1) DELAY = 0 DO ArcMainNG(#ArcOnMoveStd, WDAT1, WP3) PRIO = -1
  ArcMainNG(#ArcOnBeforeMoveStd, WDAT1, WP3)
  LIN XP3
  ArcMainNG(#ArcOnAfterMoveStd, WDAT1, WP3)
;ENDFOLD
   $VEL.CP = 0.025
   LIN  {X -8.829, Y 8.706, Z 19.900, A 0.000, B 0.000, C 0.000} C_DIS
   $VEL.CP = 0.060
   LIN  {X -8.706, Y 8.829, Z 19.900, A 0.000, B 0.000, C 0.000} C_DIS

;FOLD ARCOFF WDAT2 LIN P4 CPDAT2 Tool[1]:cmttorch Base[1]:vrashatel ;%{PE}
  ;FOLD Parameters ;%{h}
    ;Params IlfProvider=kukaroboter.arctech.arcofflin; Kuka.IsGlobalPoint=False; Kuka.PointName=P4; Kuka.BlendingEnabled=False; Kuka.MoveDataName=CPDAT2; Kuka.VelocityPath=0.01; Kuka.CurrentCDSetIndex=0; Kuka.MovementParameterFieldEnabled=True; ArcTech.WdatVarName=WDAT2; ArcTech.Basic=3.4.3.1264
  ;ENDFOLD
  $BWDSTART = FALSE
  LDAT_ACT = LCPDAT2
  FDAT_ACT = FP4
  BAS(#CP_PARAMS, gArcBasVelDefinition)
  SET_CD_PARAMS (0)
  TRIGGER WHEN PATH = ArcGetPath(#ArcOffBefore, WDAT2) DELAY = 0 DO ArcMainNG(#ArcOffBeforeOffStd, WDAT2, WP4) PRIO = -1
  TRIGGER WHEN PATH = ArcGetPath(#OnTheFlyArcOff, WDAT2) DELAY = 0 DO ArcMainNG(#ArcOffMoveStd, WDAT2, WP4) PRIO = -1
  ArcMainNG(#ArcOffBeforeMoveStd, WDAT2, WP4)
  LIN XP4
  ArcMainNG(#ArcOffAfterMoveStd, WDAT2, WP4)
;ENDFOLD
   $VEL.CP = 0.080
   LIN  {X -8.140, Y 8.829, Z 19.900, A 0.000, B 0.000, C 0.000} C_DIS

;FOLD ARCON WDAT1 LIN P3 Vel=0.5 m/s CPDAT1 Tool[1]:cmttorch Base[1]:vrashatel ;%{PE}
  ;FOLD Parameters ;%{h}
    ;Params IlfProvider=kukaroboter.arctech.arconlin; Kuka.IsGlobalPoint=False; Kuka.PointName=P3; Kuka.BlendingEnabled=False; Kuka.MoveDataName=CPDAT1; Kuka.VelocityPath=0.5; Kuka.CurrentCDSetIndex=0; Kuka.MovementParameterFieldEnabled=True; ArcTech.WdatVarName=WDAT1; ArcTech.Basic=3.4.3.1264
  ;ENDFOLD
  $BWDSTART = FALSE
  LDAT_ACT = LCPDAT1
  FDAT_ACT = FP3
  BAS(#CP_PARAMS, 0.5)
  SET_CD_PARAMS (0)
  TRIGGER WHEN DISTANCE = 1 DELAY = ArcGetDelay(#PreDefinition, WDAT1) DO ArcMainNG(#PreDefinition, WDAT1, WP3) PRIO = -1
  TRIGGER WHEN PATH = ArcGetPath(#OnTheFlyArcOn, WDAT1) DELAY = ArcGetDelay(#GasPreflow, WDAT1) DO ArcMainNG(#GasPreflow, WDAT1, WP3) PRIO = -1
  TRIGGER WHEN PATH = ArcGetPath(#OnTheFlyArcOn, WDAT1) DELAY = 0 DO ArcMainNG(#ArcOnMoveStd, WDAT1, WP3) PRIO = -1
  ArcMainNG(#ArcOnBeforeMoveStd, WDAT1, WP3)
  LIN XP3
  ArcMainNG(#ArcOnAfterMoveStd, WDAT1, WP3)
;ENDFOLD
   $VEL.CP = 0.060
   LIN  {X -8.829, Y 8.140, Z 19.900, A 0.000, B 0.000, C 0.000} C_DIS

;FOLD ARCOFF WDAT2 LIN P4 CPDAT2 Tool[1]:cmttorch Base[1]:vrashatel ;%{PE}
  ;FOLD Parameters ;%{h}
    ;Params IlfProvider=kukaroboter.arctech.arcofflin; Kuka.IsGlobalPoint=False; Kuka.PointName=P4; Kuka.BlendingEnabled=False; Kuka.MoveDataName=CPDAT2; Kuka.VelocityPath=0.01; Kuka.CurrentCDSetIndex=0; Kuka.MovementParameterFieldEnabled=True; ArcTech.WdatVarName=WDAT2; ArcTech.Basic=3.4.3.1264
  ;ENDFOLD
  $BWDSTART = FALSE
  LDAT_ACT = LCPDAT2
  FDAT_ACT = FP4
  BAS(#CP_PARAMS, gArcBasVelDefinition)
  SET_CD_PARAMS (0)
  TRIGGER WHEN PATH = ArcGetPath(#ArcOffBefore, WDAT2) DELAY = 0 DO ArcMainNG(#ArcOffBeforeOffStd, WDAT2, WP4) PRIO = -1
  TRIGGER WHEN PATH = ArcGetPath(#OnTheFlyArcOff, WDAT2) DELAY = 0 DO ArcMainNG(#ArcOffMoveStd, WDAT2, WP4) PRIO = -1
  ArcMainNG(#ArcOffBeforeMoveStd, WDAT2, WP4)
  LIN XP4
  ArcMainNG(#ArcOffAfterMoveStd, WDAT2, WP4)
;ENDFOLD
   $VEL.CP = 0.080
   LIN  {X -8.829, Y 7.575, Z 19.900, A 0.000, B 0.000, C 0.000} C_DIS

;FOLD ARCON WDAT1 LIN P3 Vel=0.5 m/s CPDAT1 Tool[1]:cmttorch Base[1]:vrashatel ;%{PE}
  ;FOLD Parameters ;%{h}
    ;Params IlfProvider=kukaroboter.arctech.arconlin; Kuka.IsGlobalPoint=False; Kuka.PointName=P3; Kuka.BlendingEnabled=False; Kuka.MoveDataName=CPDAT1; Kuka.VelocityPath=0.5; Kuka.CurrentCDSetIndex=0; Kuka.MovementParameterFieldEnabled=True; ArcTech.WdatVarName=WDAT1; ArcTech.Basic=3.4.3.1264
  ;ENDFOLD
  $BWDSTART = FALSE
  LDAT_ACT = LCPDAT1
  FDAT_ACT = FP3
  BAS(#CP_PARAMS, 0.5)
  SET_CD_PARAMS (0)
  TRIGGER WHEN DISTANCE = 1 DELAY = ArcGetDelay(#PreDefinition, WDAT1) DO ArcMainNG(#PreDefinition, WDAT1, WP3) PRIO = -1
  TRIGGER WHEN PATH = ArcGetPath(#OnTheFlyArcOn, WDAT1) DELAY = ArcGetDelay(#GasPreflow, WDAT1) DO ArcMainNG(#GasPreflow, WDAT1, WP3) PRIO = -1
  TRIGGER WHEN PATH = ArcGetPath(#OnTheFlyArcOn, WDAT1) DELAY = 0 DO ArcMainNG(#ArcOnMoveStd, WDAT1, WP3) PRIO = -1
  ArcMainNG(#ArcOnBeforeMoveStd, WDAT1, WP3)
  LIN XP3
  ArcMainNG(#ArcOnAfterMoveStd, WDAT1, WP3)
;ENDFOLD
   $VEL.CP = 0.060
   LIN  {X -7.575, Y 8.829, Z 19.900, A 0.000, B 0.000, C 0.000} C_DIS

;FOLD ARCOFF WDAT2 LIN P4 CPDAT2 Tool[1]:cmttorch Base[1]:vrashatel ;%{PE}
  ;FOLD Parameters ;%{h}
    ;Params IlfProvider=kukaroboter.arctech.arcofflin; Kuka.IsGlobalPoint=False; Kuka.PointName=P4; Kuka.BlendingEnabled=False; Kuka.MoveDataName=CPDAT2; Kuka.VelocityPath=0.01; Kuka.CurrentCDSetIndex=0; Kuka.MovementParameterFieldEnabled=True; ArcTech.WdatVarName=WDAT2; ArcTech.Basic=3.4.3.1264
  ;ENDFOLD
  $BWDSTART = FALSE
  LDAT_ACT = LCPDAT2
  FDAT_ACT = FP4
  BAS(#CP_PARAMS, gArcBasVelDefinition)
  SET_CD_PARAMS (0)
  TRIGGER WHEN PATH = ArcGetPath(#ArcOffBefore, WDAT2) DELAY = 0 DO ArcMainNG(#ArcOffBeforeOffStd, WDAT2, WP4) PRIO = -1
  TRIGGER WHEN PATH = ArcGetPath(#OnTheFlyArcOff, WDAT2) DELAY = 0 DO ArcMainNG(#ArcOffMoveStd, WDAT2, WP4) PRIO = -1
  ArcMainNG(#ArcOffBeforeMoveStd, WDAT2, WP4)
  LIN XP4
  ArcMainNG(#ArcOffAfterMoveStd, WDAT2, WP4)
;ENDFOLD
   $VEL.CP = 0.080
   LIN  {X -7.009, Y 8.829, Z 19.900, A 0.000, B 0.000, C 0.000} C_DIS

;FOLD ARCON WDAT1 LIN P3 Vel=0.5 m/s CPDAT1 Tool[1]:cmttorch Base[1]:vrashatel ;%{PE}
  ;FOLD Parameters ;%{h}
    ;Params IlfProvider=kukaroboter.arctech.arconlin; Kuka.IsGlobalPoint=False; Kuka.PointName=P3; Kuka.BlendingEnabled=False; Kuka.MoveDataName=CPDAT1; Kuka.VelocityPath=0.5; Kuka.CurrentCDSetIndex=0; Kuka.MovementParameterFieldEnabled=True; ArcTech.WdatVarName=WDAT1; ArcTech.Basic=3.4.3.1264
  ;ENDFOLD
  $BWDSTART = FALSE
  LDAT_ACT = LCPDAT1
  FDAT_ACT = FP3
  BAS(#CP_PARAMS, 0.5)
  SET_CD_PARAMS (0)
  TRIGGER WHEN DISTANCE = 1 DELAY = ArcGetDelay(#PreDefinition, WDAT1) DO ArcMainNG(#PreDefinition, WDAT1, WP3) PRIO = -1
  TRIGGER WHEN PATH = ArcGetPath(#OnTheFlyArcOn, WDAT1) DELAY = ArcGetDelay(#GasPreflow, WDAT1) DO ArcMainNG(#GasPreflow, WDAT1, WP3) PRIO = -1
  TRIGGER WHEN PATH = ArcGetPath(#OnTheFlyArcOn, WDAT1) DELAY = 0 DO ArcMainNG(#ArcOnMoveStd, WDAT1, WP3) PRIO = -1
  ArcMainNG(#ArcOnBeforeMoveStd, WDAT1, WP3)
  LIN XP3
  ArcMainNG(#ArcOnAfterMoveStd, WDAT1, WP3)
;ENDFOLD
   $VEL.CP = 0.060
   LIN  {X -8.829, Y 7.009, Z 19.900, A 0.000, B 0.000, C 0.000} C_DIS

;FOLD ARCOFF WDAT2 LIN P4 CPDAT2 Tool[1]:cmttorch Base[1]:vrashatel ;%{PE}
  ;FOLD Parameters ;%{h}
    ;Params IlfProvider=kukaroboter.arctech.arcofflin; Kuka.IsGlobalPoint=False; Kuka.PointName=P4; Kuka.BlendingEnabled=False; Kuka.MoveDataName=CPDAT2; Kuka.VelocityPath=0.01; Kuka.CurrentCDSetIndex=0; Kuka.MovementParameterFieldEnabled=True; ArcTech.WdatVarName=WDAT2; ArcTech.Basic=3.4.3.1264
  ;ENDFOLD
  $BWDSTART = FALSE
  LDAT_ACT = LCPDAT2
  FDAT_ACT = FP4
  BAS(#CP_PARAMS, gArcBasVelDefinition)
  SET_CD_PARAMS (0)
  TRIGGER WHEN PATH = ArcGetPath(#ArcOffBefore, WDAT2) DELAY = 0 DO ArcMainNG(#ArcOffBeforeOffStd, WDAT2, WP4) PRIO = -1
  TRIGGER WHEN PATH = ArcGetPath(#OnTheFlyArcOff, WDAT2) DELAY = 0 DO ArcMainNG(#ArcOffMoveStd, WDAT2, WP4) PRIO = -1
  ArcMainNG(#ArcOffBeforeMoveStd, WDAT2, WP4)
  LIN XP4
  ArcMainNG(#ArcOffAfterMoveStd, WDAT2, WP4)
;ENDFOLD
   $VEL.CP = 0.080
   LIN  {X -8.829, Y 6.443, Z 19.900, A 0.000, B 0.000, C 0.000} C_DIS

;FOLD ARCON WDAT1 LIN P3 Vel=0.5 m/s CPDAT1 Tool[1]:cmttorch Base[1]:vrashatel ;%{PE}
  ;FOLD Parameters ;%{h}
    ;Params IlfProvider=kukaroboter.arctech.arconlin; Kuka.IsGlobalPoint=False; Kuka.PointName=P3; Kuka.BlendingEnabled=False; Kuka.MoveDataName=CPDAT1; Kuka.VelocityPath=0.5; Kuka.CurrentCDSetIndex=0; Kuka.MovementParameterFieldEnabled=True; ArcTech.WdatVarName=WDAT1; ArcTech.Basic=3.4.3.1264
  ;ENDFOLD
  $BWDSTART = FALSE
  LDAT_ACT = LCPDAT1
  FDAT_ACT = FP3
  BAS(#CP_PARAMS, 0.5)
  SET_CD_PARAMS (0)
  TRIGGER WHEN DISTANCE = 1 DELAY = ArcGetDelay(#PreDefinition, WDAT1) DO ArcMainNG(#PreDefinition, WDAT1, WP3) PRIO = -1
  TRIGGER WHEN PATH = ArcGetPath(#OnTheFlyArcOn, WDAT1) DELAY = ArcGetDelay(#GasPreflow, WDAT1) DO ArcMainNG(#GasPreflow, WDAT1, WP3) PRIO = -1
  TRIGGER WHEN PATH = ArcGetPath(#OnTheFlyArcOn, WDAT1) DELAY = 0 DO ArcMainNG(#ArcOnMoveStd, WDAT1, WP3) PRIO = -1
  ArcMainNG(#ArcOnBeforeMoveStd, WDAT1, WP3)
  LIN XP3
  ArcMainNG(#ArcOnAfterMoveStd, WDAT1, WP3)
;ENDFOLD
   $VEL.CP = 0.060
   LIN  {X -6.443, Y 8.829, Z 19.900, A 0.000, B 0.000, C 0.000} C_DIS

;FOLD ARCOFF WDAT2 LIN P4 CPDAT2 Tool[1]:cmttorch Base[1]:vrashatel ;%{PE}
  ;FOLD Parameters ;%{h}
    ;Params IlfProvider=kukaroboter.arctech.arcofflin; Kuka.IsGlobalPoint=False; Kuka.PointName=P4; Kuka.BlendingEnabled=False; Kuka.MoveDataName=CPDAT2; Kuka.VelocityPath=0.01; Kuka.CurrentCDSetIndex=0; Kuka.MovementParameterFieldEnabled=True; ArcTech.WdatVarName=WDAT2; ArcTech.Basic=3.4.3.1264
  ;ENDFOLD
  $BWDSTART = FALSE
  LDAT_ACT = LCPDAT2
  FDAT_ACT = FP4
  BAS(#CP_PARAMS, gArcBasVelDefinition)
  SET_CD_PARAMS (0)
  TRIGGER WHEN PATH = ArcGetPath(#ArcOffBefore, WDAT2) DELAY = 0 DO ArcMainNG(#ArcOffBeforeOffStd, WDAT2, WP4) PRIO = -1
  TRIGGER WHEN PATH = ArcGetPath(#OnTheFlyArcOff, WDAT2) DELAY = 0 DO ArcMainNG(#ArcOffMoveStd, WDAT2, WP4) PRIO = -1
  ArcMainNG(#ArcOffBeforeMoveStd, WDAT2, WP4)
  LIN XP4
  ArcMainNG(#ArcOffAfterMoveStd, WDAT2, WP4)
;ENDFOLD
   $VEL.CP = 0.080
   LIN  {X -5.878, Y 8.829, Z 19.900, A 0.000, B 0.000, C 0.000} C_DIS

;FOLD ARCON WDAT1 LIN P3 Vel=0.5 m/s CPDAT1 Tool[1]:cmttorch Base[1]:vrashatel ;%{PE}
  ;FOLD Parameters ;%{h}
    ;Params IlfProvider=kukaroboter.arctech.arconlin; Kuka.IsGlobalPoint=False; Kuka.PointName=P3; Kuka.BlendingEnabled=False; Kuka.MoveDataName=CPDAT1; Kuka.VelocityPath=0.5; Kuka.CurrentCDSetIndex=0; Kuka.MovementParameterFieldEnabled=True; ArcTech.WdatVarName=WDAT1; ArcTech.Basic=3.4.3.1264
  ;ENDFOLD
  $BWDSTART = FALSE
  LDAT_ACT = LCPDAT1
  FDAT_ACT = FP3
  BAS(#CP_PARAMS, 0.5)
  SET_CD_PARAMS (0)
  TRIGGER WHEN DISTANCE = 1 DELAY = ArcGetDelay(#PreDefinition, WDAT1) DO ArcMainNG(#PreDefinition, WDAT1, WP3) PRIO = -1
  TRIGGER WHEN PATH = ArcGetPath(#OnTheFlyArcOn, WDAT1) DELAY = ArcGetDelay(#GasPreflow, WDAT1) DO ArcMainNG(#GasPreflow, WDAT1, WP3) PRIO = -1
  TRIGGER WHEN PATH = ArcGetPath(#OnTheFlyArcOn, WDAT1) DELAY = 0 DO ArcMainNG(#ArcOnMoveStd, WDAT1, WP3) PRIO = -1
  ArcMainNG(#ArcOnBeforeMoveStd, WDAT1, WP3)
  LIN XP3
  ArcMainNG(#ArcOnAfterMoveStd, WDAT1, WP3)
;ENDFOLD
   $VEL.CP = 0.060
   LIN  {X -8.829, Y 5.878, Z 19.900, A 0.000, B 0.000, C 0.000} C_DIS

;FOLD ARCOFF WDAT2 LIN P4 CPDAT2 Tool[1]:cmttorch Base[1]:vrashatel ;%{PE}
  ;FOLD Parameters ;%{h}
    ;Params IlfProvider=kukaroboter.arctech.arcofflin; Kuka.IsGlobalPoint=False; Kuka.PointName=P4; Kuka.BlendingEnabled=False; Kuka.MoveDataName=CPDAT2; Kuka.VelocityPath=0.01; Kuka.CurrentCDSetIndex=0; Kuka.MovementParameterFieldEnabled=True; ArcTech.WdatVarName=WDAT2; ArcTech.Basic=3.4.3.1264
  ;ENDFOLD
  $BWDSTART = FALSE
  LDAT_ACT = LCPDAT2
  FDAT_ACT = FP4
  BAS(#CP_PARAMS, gArcBasVelDefinition)
  SET_CD_PARAMS (0)
  TRIGGER WHEN PATH = ArcGetPath(#ArcOffBefore, WDAT2) DELAY = 0 DO ArcMainNG(#ArcOffBeforeOffStd, WDAT2, WP4) PRIO = -1
  TRIGGER WHEN PATH = ArcGetPath(#OnTheFlyArcOff, WDAT2) DELAY = 0 DO ArcMainNG(#ArcOffMoveStd, WDAT2, WP4) PRIO = -1
  ArcMainNG(#ArcOffBeforeMoveStd, WDAT2, WP4)
  LIN XP4
  ArcMainNG(#ArcOffAfterMoveStd, WDAT2, WP4)
;ENDFOLD
   $VEL.CP = 0.080
   LIN  {X -8.829, Y 5.312, Z 19.900, A 0.000, B 0.000, C 0.000} C_DIS

;FOLD ARCON WDAT1 LIN P3 Vel=0.5 m/s CPDAT1 Tool[1]:cmttorch Base[1]:vrashatel ;%{PE}
  ;FOLD Parameters ;%{h}
    ;Params IlfProvider=kukaroboter.arctech.arconlin; Kuka.IsGlobalPoint=False; Kuka.PointName=P3; Kuka.BlendingEnabled=False; Kuka.MoveDataName=CPDAT1; Kuka.VelocityPath=0.5; Kuka.CurrentCDSetIndex=0; Kuka.MovementParameterFieldEnabled=True; ArcTech.WdatVarName=WDAT1; ArcTech.Basic=3.4.3.1264
  ;ENDFOLD
  $BWDSTART = FALSE
  LDAT_ACT = LCPDAT1
  FDAT_ACT = FP3
  BAS(#CP_PARAMS, 0.5)
  SET_CD_PARAMS (0)
  TRIGGER WHEN DISTANCE = 1 DELAY = ArcGetDelay(#PreDefinition, WDAT1) DO ArcMainNG(#PreDefinition, WDAT1, WP3) PRIO = -1
  TRIGGER WHEN PATH = ArcGetPath(#OnTheFlyArcOn, WDAT1) DELAY = ArcGetDelay(#GasPreflow, WDAT1) DO ArcMainNG(#GasPreflow, WDAT1, WP3) PRIO = -1
  TRIGGER WHEN PATH = ArcGetPath(#OnTheFlyArcOn, WDAT1) DELAY = 0 DO ArcMainNG(#ArcOnMoveStd, WDAT1, WP3) PRIO = -1
  ArcMainNG(#ArcOnBeforeMoveStd, WDAT1, WP3)
  LIN XP3
  ArcMainNG(#ArcOnAfterMoveStd, WDAT1, WP3)
;ENDFOLD
   $VEL.CP = 0.060
   LIN  {X -5.312, Y 8.829, Z 19.900, A 0.000, B 0.000, C 0.000} C_DIS

;FOLD ARCOFF WDAT2 LIN P4 CPDAT2 Tool[1]:cmttorch Base[1]:vrashatel ;%{PE}
  ;FOLD Parameters ;%{h}
    ;Params IlfProvider=kukaroboter.arctech.arcofflin; Kuka.IsGlobalPoint=False; Kuka.PointName=P4; Kuka.BlendingEnabled=False; Kuka.MoveDataName=CPDAT2; Kuka.VelocityPath=0.01; Kuka.CurrentCDSetIndex=0; Kuka.MovementParameterFieldEnabled=True; ArcTech.WdatVarName=WDAT2; ArcTech.Basic=3.4.3.1264
  ;ENDFOLD
  $BWDSTART = FALSE
  LDAT_ACT = LCPDAT2
  FDAT_ACT = FP4
  BAS(#CP_PARAMS, gArcBasVelDefinition)
  SET_CD_PARAMS (0)
  TRIGGER WHEN PATH = ArcGetPath(#ArcOffBefore, WDAT2) DELAY = 0 DO ArcMainNG(#ArcOffBeforeOffStd, WDAT2, WP4) PRIO = -1
  TRIGGER WHEN PATH = ArcGetPath(#OnTheFlyArcOff, WDAT2) DELAY = 0 DO ArcMainNG(#ArcOffMoveStd, WDAT2, WP4) PRIO = -1
  ArcMainNG(#ArcOffBeforeMoveStd, WDAT2, WP4)
  LIN XP4
  ArcMainNG(#ArcOffAfterMoveStd, WDAT2, WP4)
;ENDFOLD
   $VEL.CP = 0.080
   LIN  {X -4.746, Y 8.829, Z 19.900, A 0.000, B 0.000, C 0.000} C_DIS

;FOLD ARCON WDAT1 LIN P3 Vel=0.5 m/s CPDAT1 Tool[1]:cmttorch Base[1]:vrashatel ;%{PE}
  ;FOLD Parameters ;%{h}
    ;Params IlfProvider=kukaroboter.arctech.arconlin; Kuka.IsGlobalPoint=False; Kuka.PointName=P3; Kuka.BlendingEnabled=False; Kuka.MoveDataName=CPDAT1; Kuka.VelocityPath=0.5; Kuka.CurrentCDSetIndex=0; Kuka.MovementParameterFieldEnabled=True; ArcTech.WdatVarName=WDAT1; ArcTech.Basic=3.4.3.1264
  ;ENDFOLD
  $BWDSTART = FALSE
  LDAT_ACT = LCPDAT1
  FDAT_ACT = FP3
  BAS(#CP_PARAMS, 0.5)
  SET_CD_PARAMS (0)
  TRIGGER WHEN DISTANCE = 1 DELAY = ArcGetDelay(#PreDefinition, WDAT1) DO ArcMainNG(#PreDefinition, WDAT1, WP3) PRIO = -1
  TRIGGER WHEN PATH = ArcGetPath(#OnTheFlyArcOn, WDAT1) DELAY = ArcGetDelay(#GasPreflow, WDAT1) DO ArcMainNG(#GasPreflow, WDAT1, WP3) PRIO = -1
  TRIGGER WHEN PATH = ArcGetPath(#OnTheFlyArcOn, WDAT1) DELAY = 0 DO ArcMainNG(#ArcOnMoveStd, WDAT1, WP3) PRIO = -1
  ArcMainNG(#ArcOnBeforeMoveStd, WDAT1, WP3)
  LIN XP3
  ArcMainNG(#ArcOnAfterMoveStd, WDAT1, WP3)
;ENDFOLD
   $VEL.CP = 0.060
   LIN  {X -8.829, Y 4.746, Z 19.900, A 0.000, B 0.000, C 0.000} C_DIS

;FOLD ARCOFF WDAT2 LIN P4 CPDAT2 Tool[1]:cmttorch Base[1]:vrashatel ;%{PE}
  ;FOLD Parameters ;%{h}
    ;Params IlfProvider=kukaroboter.arctech.arcofflin; Kuka.IsGlobalPoint=False; Kuka.PointName=P4; Kuka.BlendingEnabled=False; Kuka.MoveDataName=CPDAT2; Kuka.VelocityPath=0.01; Kuka.CurrentCDSetIndex=0; Kuka.MovementParameterFieldEnabled=True; ArcTech.WdatVarName=WDAT2; ArcTech.Basic=3.4.3.1264
  ;ENDFOLD
  $BWDSTART = FALSE
  LDAT_ACT = LCPDAT2
  FDAT_ACT = FP4
  BAS(#CP_PARAMS, gArcBasVelDefinition)
  SET_CD_PARAMS (0)
  TRIGGER WHEN PATH = ArcGetPath(#ArcOffBefore, WDAT2) DELAY = 0 DO ArcMainNG(#ArcOffBeforeOffStd, WDAT2, WP4) PRIO = -1
  TRIGGER WHEN PATH = ArcGetPath(#OnTheFlyArcOff, WDAT2) DELAY = 0 DO ArcMainNG(#ArcOffMoveStd, WDAT2, WP4) PRIO = -1
  ArcMainNG(#ArcOffBeforeMoveStd, WDAT2, WP4)
  LIN XP4
  ArcMainNG(#ArcOffAfterMoveStd, WDAT2, WP4)
;ENDFOLD
   $VEL.CP = 0.080
   LIN  {X -8.829, Y 4.181, Z 19.900, A 0.000, B 0.000, C 0.000} C_DIS

;FOLD ARCON WDAT1 LIN P3 Vel=0.5 m/s CPDAT1 Tool[1]:cmttorch Base[1]:vrashatel ;%{PE}
  ;FOLD Parameters ;%{h}
    ;Params IlfProvider=kukaroboter.arctech.arconlin; Kuka.IsGlobalPoint=False; Kuka.PointName=P3; Kuka.BlendingEnabled=False; Kuka.MoveDataName=CPDAT1; Kuka.VelocityPath=0.5; Kuka.CurrentCDSetIndex=0; Kuka.MovementParameterFieldEnabled=True; ArcTech.WdatVarName=WDAT1; ArcTech.Basic=3.4.3.1264
  ;ENDFOLD
  $BWDSTART = FALSE
  LDAT_ACT = LCPDAT1
  FDAT_ACT = FP3
  BAS(#CP_PARAMS, 0.5)
  SET_CD_PARAMS (0)
  TRIGGER WHEN DISTANCE = 1 DELAY = ArcGetDelay(#PreDefinition, WDAT1) DO ArcMainNG(#PreDefinition, WDAT1, WP3) PRIO = -1
  TRIGGER WHEN PATH = ArcGetPath(#OnTheFlyArcOn, WDAT1) DELAY = ArcGetDelay(#GasPreflow, WDAT1) DO ArcMainNG(#GasPreflow, WDAT1, WP3) PRIO = -1
  TRIGGER WHEN PATH = ArcGetPath(#OnTheFlyArcOn, WDAT1) DELAY = 0 DO ArcMainNG(#ArcOnMoveStd, WDAT1, WP3) PRIO = -1
  ArcMainNG(#ArcOnBeforeMoveStd, WDAT1, WP3)
  LIN XP3
  ArcMainNG(#ArcOnAfterMoveStd, WDAT1, WP3)
;ENDFOLD
   $VEL.CP = 0.060
   LIN  {X -4.181, Y 8.829, Z 19.900, A 0.000, B 0.000, C 0.000} C_DIS

;FOLD ARCOFF WDAT2 LIN P4 CPDAT2 Tool[1]:cmttorch Base[1]:vrashatel ;%{PE}
  ;FOLD Parameters ;%{h}
    ;Params IlfProvider=kukaroboter.arctech.arcofflin; Kuka.IsGlobalPoint=False; Kuka.PointName=P4; Kuka.BlendingEnabled=False; Kuka.MoveDataName=CPDAT2; Kuka.VelocityPath=0.01; Kuka.CurrentCDSetIndex=0; Kuka.MovementParameterFieldEnabled=True; ArcTech.WdatVarName=WDAT2; ArcTech.Basic=3.4.3.1264
  ;ENDFOLD
  $BWDSTART = FALSE
  LDAT_ACT = LCPDAT2
  FDAT_ACT = FP4
  BAS(#CP_PARAMS, gArcBasVelDefinition)
  SET_CD_PARAMS (0)
  TRIGGER WHEN PATH = ArcGetPath(#ArcOffBefore, WDAT2) DELAY = 0 DO ArcMainNG(#ArcOffBeforeOffStd, WDAT2, WP4) PRIO = -1
  TRIGGER WHEN PATH = ArcGetPath(#OnTheFlyArcOff, WDAT2) DELAY = 0 DO ArcMainNG(#ArcOffMoveStd, WDAT2, WP4) PRIO = -1
  ArcMainNG(#ArcOffBeforeMoveStd, WDAT2, WP4)
  LIN XP4
  ArcMainNG(#ArcOffAfterMoveStd, WDAT2, WP4)
;ENDFOLD
   $VEL.CP = 0.080
   LIN  {X -3.615, Y 8.829, Z 19.900, A 0.000, B 0.000, C 0.000} C_DIS

;FOLD ARCON WDAT1 LIN P3 Vel=0.5 m/s CPDAT1 Tool[1]:cmttorch Base[1]:vrashatel ;%{PE}
  ;FOLD Parameters ;%{h}
    ;Params IlfProvider=kukaroboter.arctech.arconlin; Kuka.IsGlobalPoint=False; Kuka.PointName=P3; Kuka.BlendingEnabled=False; Kuka.MoveDataName=CPDAT1; Kuka.VelocityPath=0.5; Kuka.CurrentCDSetIndex=0; Kuka.MovementParameterFieldEnabled=True; ArcTech.WdatVarName=WDAT1; ArcTech.Basic=3.4.3.1264
  ;ENDFOLD
  $BWDSTART = FALSE
  LDAT_ACT = LCPDAT1
  FDAT_ACT = FP3
  BAS(#CP_PARAMS, 0.5)
  SET_CD_PARAMS (0)
  TRIGGER WHEN DISTANCE = 1 DELAY = ArcGetDelay(#PreDefinition, WDAT1) DO ArcMainNG(#PreDefinition, WDAT1, WP3) PRIO = -1
  TRIGGER WHEN PATH = ArcGetPath(#OnTheFlyArcOn, WDAT1) DELAY = ArcGetDelay(#GasPreflow, WDAT1) DO ArcMainNG(#GasPreflow, WDAT1, WP3) PRIO = -1
  TRIGGER WHEN PATH = ArcGetPath(#OnTheFlyArcOn, WDAT1) DELAY = 0 DO ArcMainNG(#ArcOnMoveStd, WDAT1, WP3) PRIO = -1
  ArcMainNG(#ArcOnBeforeMoveStd, WDAT1, WP3)
  LIN XP3
  ArcMainNG(#ArcOnAfterMoveStd, WDAT1, WP3)
;ENDFOLD
   $VEL.CP = 0.060
   LIN  {X -8.829, Y 3.615, Z 19.900, A 0.000, B 0.000, C 0.000} C_DIS

;FOLD ARCOFF WDAT2 LIN P4 CPDAT2 Tool[1]:cmttorch Base[1]:vrashatel ;%{PE}
  ;FOLD Parameters ;%{h}
    ;Params IlfProvider=kukaroboter.arctech.arcofflin; Kuka.IsGlobalPoint=False; Kuka.PointName=P4; Kuka.BlendingEnabled=False; Kuka.MoveDataName=CPDAT2; Kuka.VelocityPath=0.01; Kuka.CurrentCDSetIndex=0; Kuka.MovementParameterFieldEnabled=True; ArcTech.WdatVarName=WDAT2; ArcTech.Basic=3.4.3.1264
  ;ENDFOLD
  $BWDSTART = FALSE
  LDAT_ACT = LCPDAT2
  FDAT_ACT = FP4
  BAS(#CP_PARAMS, gArcBasVelDefinition)
  SET_CD_PARAMS (0)
  TRIGGER WHEN PATH = ArcGetPath(#ArcOffBefore, WDAT2) DELAY = 0 DO ArcMainNG(#ArcOffBeforeOffStd, WDAT2, WP4) PRIO = -1
  TRIGGER WHEN PATH = ArcGetPath(#OnTheFlyArcOff, WDAT2) DELAY = 0 DO ArcMainNG(#ArcOffMoveStd, WDAT2, WP4) PRIO = -1
  ArcMainNG(#ArcOffBeforeMoveStd, WDAT2, WP4)
  LIN XP4
  ArcMainNG(#ArcOffAfterMoveStd, WDAT2, WP4)
;ENDFOLD
   $VEL.CP = 0.080
   LIN  {X -8.829, Y 3.049, Z 19.900, A 0.000, B 0.000, C 0.000} C_DIS

;FOLD ARCON WDAT1 LIN P3 Vel=0.5 m/s CPDAT1 Tool[1]:cmttorch Base[1]:vrashatel ;%{PE}
  ;FOLD Parameters ;%{h}
    ;Params IlfProvider=kukaroboter.arctech.arconlin; Kuka.IsGlobalPoint=False; Kuka.PointName=P3; Kuka.BlendingEnabled=False; Kuka.MoveDataName=CPDAT1; Kuka.VelocityPath=0.5; Kuka.CurrentCDSetIndex=0; Kuka.MovementParameterFieldEnabled=True; ArcTech.WdatVarName=WDAT1; ArcTech.Basic=3.4.3.1264
  ;ENDFOLD
  $BWDSTART = FALSE
  LDAT_ACT = LCPDAT1
  FDAT_ACT = FP3
  BAS(#CP_PARAMS, 0.5)
  SET_CD_PARAMS (0)
  TRIGGER WHEN DISTANCE = 1 DELAY = ArcGetDelay(#PreDefinition, WDAT1) DO ArcMainNG(#PreDefinition, WDAT1, WP3) PRIO = -1
  TRIGGER WHEN PATH = ArcGetPath(#OnTheFlyArcOn, WDAT1) DELAY = ArcGetDelay(#GasPreflow, WDAT1) DO ArcMainNG(#GasPreflow, WDAT1, WP3) PRIO = -1
  TRIGGER WHEN PATH = ArcGetPath(#OnTheFlyArcOn, WDAT1) DELAY = 0 DO ArcMainNG(#ArcOnMoveStd, WDAT1, WP3) PRIO = -1
  ArcMainNG(#ArcOnBeforeMoveStd, WDAT1, WP3)
  LIN XP3
  ArcMainNG(#ArcOnAfterMoveStd, WDAT1, WP3)
;ENDFOLD
   $VEL.CP = 0.060
   LIN  {X -4.763, Y 7.116, Z 19.900, A 0.000, B 0.000, C 0.000} C_DIS

;FOLD ARCOFF WDAT2 LIN P4 CPDAT2 Tool[1]:cmttorch Base[1]:vrashatel ;%{PE}
  ;FOLD Parameters ;%{h}
    ;Params IlfProvider=kukaroboter.arctech.arcofflin; Kuka.IsGlobalPoint=False; Kuka.PointName=P4; Kuka.BlendingEnabled=False; Kuka.MoveDataName=CPDAT2; Kuka.VelocityPath=0.01; Kuka.CurrentCDSetIndex=0; Kuka.MovementParameterFieldEnabled=True; ArcTech.WdatVarName=WDAT2; ArcTech.Basic=3.4.3.1264
  ;ENDFOLD
  $BWDSTART = FALSE
  LDAT_ACT = LCPDAT2
  FDAT_ACT = FP4
  BAS(#CP_PARAMS, gArcBasVelDefinition)
  SET_CD_PARAMS (0)
  TRIGGER WHEN PATH = ArcGetPath(#ArcOffBefore, WDAT2) DELAY = 0 DO ArcMainNG(#ArcOffBeforeOffStd, WDAT2, WP4) PRIO = -1
  TRIGGER WHEN PATH = ArcGetPath(#OnTheFlyArcOff, WDAT2) DELAY = 0 DO ArcMainNG(#ArcOffMoveStd, WDAT2, WP4) PRIO = -1
  ArcMainNG(#ArcOffBeforeMoveStd, WDAT2, WP4)
  LIN XP4
  ArcMainNG(#ArcOffAfterMoveStd, WDAT2, WP4)
;ENDFOLD
   $VEL.CP = 0.080
   LIN  {X -4.391, Y 7.487, Z 19.900, A 0.000, B 0.000, C 0.000} C_DIS

;FOLD ARCON WDAT1 LIN P3 Vel=0.5 m/s CPDAT1 Tool[1]:cmttorch Base[1]:vrashatel ;%{PE}
  ;FOLD Parameters ;%{h}
    ;Params IlfProvider=kukaroboter.arctech.arconlin; Kuka.IsGlobalPoint=False; Kuka.PointName=P3; Kuka.BlendingEnabled=False; Kuka.MoveDataName=CPDAT1; Kuka.VelocityPath=0.5; Kuka.CurrentCDSetIndex=0; Kuka.MovementParameterFieldEnabled=True; ArcTech.WdatVarName=WDAT1; ArcTech.Basic=3.4.3.1264
  ;ENDFOLD
  $BWDSTART = FALSE
  LDAT_ACT = LCPDAT1
  FDAT_ACT = FP3
  BAS(#CP_PARAMS, 0.5)
  SET_CD_PARAMS (0)
  TRIGGER WHEN DISTANCE = 1 DELAY = ArcGetDelay(#PreDefinition, WDAT1) DO ArcMainNG(#PreDefinition, WDAT1, WP3) PRIO = -1
  TRIGGER WHEN PATH = ArcGetPath(#OnTheFlyArcOn, WDAT1) DELAY = ArcGetDelay(#GasPreflow, WDAT1) DO ArcMainNG(#GasPreflow, WDAT1, WP3) PRIO = -1
  TRIGGER WHEN PATH = ArcGetPath(#OnTheFlyArcOn, WDAT1) DELAY = 0 DO ArcMainNG(#ArcOnMoveStd, WDAT1, WP3) PRIO = -1
  ArcMainNG(#ArcOnBeforeMoveStd, WDAT1, WP3)
  LIN XP3
  ArcMainNG(#ArcOnAfterMoveStd, WDAT1, WP3)
;ENDFOLD
   $VEL.CP = 0.060
   LIN  {X -3.049, Y 8.829, Z 19.900, A 0.000, B 0.000, C 0.000} C_DIS

;FOLD ARCOFF WDAT2 LIN P4 CPDAT2 Tool[1]:cmttorch Base[1]:vrashatel ;%{PE}
  ;FOLD Parameters ;%{h}
    ;Params IlfProvider=kukaroboter.arctech.arcofflin; Kuka.IsGlobalPoint=False; Kuka.PointName=P4; Kuka.BlendingEnabled=False; Kuka.MoveDataName=CPDAT2; Kuka.VelocityPath=0.01; Kuka.CurrentCDSetIndex=0; Kuka.MovementParameterFieldEnabled=True; ArcTech.WdatVarName=WDAT2; ArcTech.Basic=3.4.3.1264
  ;ENDFOLD
  $BWDSTART = FALSE
  LDAT_ACT = LCPDAT2
  FDAT_ACT = FP4
  BAS(#CP_PARAMS, gArcBasVelDefinition)
  SET_CD_PARAMS (0)
  TRIGGER WHEN PATH = ArcGetPath(#ArcOffBefore, WDAT2) DELAY = 0 DO ArcMainNG(#ArcOffBeforeOffStd, WDAT2, WP4) PRIO = -1
  TRIGGER WHEN PATH = ArcGetPath(#OnTheFlyArcOff, WDAT2) DELAY = 0 DO ArcMainNG(#ArcOffMoveStd, WDAT2, WP4) PRIO = -1
  ArcMainNG(#ArcOffBeforeMoveStd, WDAT2, WP4)
  LIN XP4
  ArcMainNG(#ArcOffAfterMoveStd, WDAT2, WP4)
;ENDFOLD
   $VEL.CP = 0.080
   LIN  {X -2.484, Y 8.829, Z 19.900, A 0.000, B 0.000, C 0.000} C_DIS

;FOLD ARCON WDAT1 LIN P3 Vel=0.5 m/s CPDAT1 Tool[1]:cmttorch Base[1]:vrashatel ;%{PE}
  ;FOLD Parameters ;%{h}
    ;Params IlfProvider=kukaroboter.arctech.arconlin; Kuka.IsGlobalPoint=False; Kuka.PointName=P3; Kuka.BlendingEnabled=False; Kuka.MoveDataName=CPDAT1; Kuka.VelocityPath=0.5; Kuka.CurrentCDSetIndex=0; Kuka.MovementParameterFieldEnabled=True; ArcTech.WdatVarName=WDAT1; ArcTech.Basic=3.4.3.1264
  ;ENDFOLD
  $BWDSTART = FALSE
  LDAT_ACT = LCPDAT1
  FDAT_ACT = FP3
  BAS(#CP_PARAMS, 0.5)
  SET_CD_PARAMS (0)
  TRIGGER WHEN DISTANCE = 1 DELAY = ArcGetDelay(#PreDefinition, WDAT1) DO ArcMainNG(#PreDefinition, WDAT1, WP3) PRIO = -1
  TRIGGER WHEN PATH = ArcGetPath(#OnTheFlyArcOn, WDAT1) DELAY = ArcGetDelay(#GasPreflow, WDAT1) DO ArcMainNG(#GasPreflow, WDAT1, WP3) PRIO = -1
  TRIGGER WHEN PATH = ArcGetPath(#OnTheFlyArcOn, WDAT1) DELAY = 0 DO ArcMainNG(#ArcOnMoveStd, WDAT1, WP3) PRIO = -1
  ArcMainNG(#ArcOnBeforeMoveStd, WDAT1, WP3)
  LIN XP3
  ArcMainNG(#ArcOnAfterMoveStd, WDAT1, WP3)
;ENDFOLD
   $VEL.CP = 0.060
   LIN  {X -3.826, Y 7.487, Z 19.900, A 0.000, B 0.000, C 0.000} C_DIS

;FOLD ARCOFF WDAT2 LIN P4 CPDAT2 Tool[1]:cmttorch Base[1]:vrashatel ;%{PE}
  ;FOLD Parameters ;%{h}
    ;Params IlfProvider=kukaroboter.arctech.arcofflin; Kuka.IsGlobalPoint=False; Kuka.PointName=P4; Kuka.BlendingEnabled=False; Kuka.MoveDataName=CPDAT2; Kuka.VelocityPath=0.01; Kuka.CurrentCDSetIndex=0; Kuka.MovementParameterFieldEnabled=True; ArcTech.WdatVarName=WDAT2; ArcTech.Basic=3.4.3.1264
  ;ENDFOLD
  $BWDSTART = FALSE
  LDAT_ACT = LCPDAT2
  FDAT_ACT = FP4
  BAS(#CP_PARAMS, gArcBasVelDefinition)
  SET_CD_PARAMS (0)
  TRIGGER WHEN PATH = ArcGetPath(#ArcOffBefore, WDAT2) DELAY = 0 DO ArcMainNG(#ArcOffBeforeOffStd, WDAT2, WP4) PRIO = -1
  TRIGGER WHEN PATH = ArcGetPath(#OnTheFlyArcOff, WDAT2) DELAY = 0 DO ArcMainNG(#ArcOffMoveStd, WDAT2, WP4) PRIO = -1
  ArcMainNG(#ArcOffBeforeMoveStd, WDAT2, WP4)
  LIN XP4
  ArcMainNG(#ArcOffAfterMoveStd, WDAT2, WP4)
;ENDFOLD
   $VEL.CP = 0.080
   LIN  {X -3.260, Y 7.487, Z 19.900, A 0.000, B 0.000, C 0.000} C_DIS

;FOLD ARCON WDAT1 LIN P3 Vel=0.5 m/s CPDAT1 Tool[1]:cmttorch Base[1]:vrashatel ;%{PE}
  ;FOLD Parameters ;%{h}
    ;Params IlfProvider=kukaroboter.arctech.arconlin; Kuka.IsGlobalPoint=False; Kuka.PointName=P3; Kuka.BlendingEnabled=False; Kuka.MoveDataName=CPDAT1; Kuka.VelocityPath=0.5; Kuka.CurrentCDSetIndex=0; Kuka.MovementParameterFieldEnabled=True; ArcTech.WdatVarName=WDAT1; ArcTech.Basic=3.4.3.1264
  ;ENDFOLD
  $BWDSTART = FALSE
  LDAT_ACT = LCPDAT1
  FDAT_ACT = FP3
  BAS(#CP_PARAMS, 0.5)
  SET_CD_PARAMS (0)
  TRIGGER WHEN DISTANCE = 1 DELAY = ArcGetDelay(#PreDefinition, WDAT1) DO ArcMainNG(#PreDefinition, WDAT1, WP3) PRIO = -1
  TRIGGER WHEN PATH = ArcGetPath(#OnTheFlyArcOn, WDAT1) DELAY = ArcGetDelay(#GasPreflow, WDAT1) DO ArcMainNG(#GasPreflow, WDAT1, WP3) PRIO = -1
  TRIGGER WHEN PATH = ArcGetPath(#OnTheFlyArcOn, WDAT1) DELAY = 0 DO ArcMainNG(#ArcOnMoveStd, WDAT1, WP3) PRIO = -1
  ArcMainNG(#ArcOnBeforeMoveStd, WDAT1, WP3)
  LIN XP3
  ArcMainNG(#ArcOnAfterMoveStd, WDAT1, WP3)
;ENDFOLD
   $VEL.CP = 0.060
   LIN  {X -1.918, Y 8.829, Z 19.900, A 0.000, B 0.000, C 0.000} C_DIS

;FOLD ARCOFF WDAT2 LIN P4 CPDAT2 Tool[1]:cmttorch Base[1]:vrashatel ;%{PE}
  ;FOLD Parameters ;%{h}
    ;Params IlfProvider=kukaroboter.arctech.arcofflin; Kuka.IsGlobalPoint=False; Kuka.PointName=P4; Kuka.BlendingEnabled=False; Kuka.MoveDataName=CPDAT2; Kuka.VelocityPath=0.01; Kuka.CurrentCDSetIndex=0; Kuka.MovementParameterFieldEnabled=True; ArcTech.WdatVarName=WDAT2; ArcTech.Basic=3.4.3.1264
  ;ENDFOLD
  $BWDSTART = FALSE
  LDAT_ACT = LCPDAT2
  FDAT_ACT = FP4
  BAS(#CP_PARAMS, gArcBasVelDefinition)
  SET_CD_PARAMS (0)
  TRIGGER WHEN PATH = ArcGetPath(#ArcOffBefore, WDAT2) DELAY = 0 DO ArcMainNG(#ArcOffBeforeOffStd, WDAT2, WP4) PRIO = -1
  TRIGGER WHEN PATH = ArcGetPath(#OnTheFlyArcOff, WDAT2) DELAY = 0 DO ArcMainNG(#ArcOffMoveStd, WDAT2, WP4) PRIO = -1
  ArcMainNG(#ArcOffBeforeMoveStd, WDAT2, WP4)
  LIN XP4
  ArcMainNG(#ArcOffAfterMoveStd, WDAT2, WP4)
;ENDFOLD
   $VEL.CP = 0.080
   LIN  {X -1.352, Y 8.829, Z 19.900, A 0.000, B 0.000, C 0.000} C_DIS

;FOLD ARCON WDAT1 LIN P3 Vel=0.5 m/s CPDAT1 Tool[1]:cmttorch Base[1]:vrashatel ;%{PE}
  ;FOLD Parameters ;%{h}
    ;Params IlfProvider=kukaroboter.arctech.arconlin; Kuka.IsGlobalPoint=False; Kuka.PointName=P3; Kuka.BlendingEnabled=False; Kuka.MoveDataName=CPDAT1; Kuka.VelocityPath=0.5; Kuka.CurrentCDSetIndex=0; Kuka.MovementParameterFieldEnabled=True; ArcTech.WdatVarName=WDAT1; ArcTech.Basic=3.4.3.1264
  ;ENDFOLD
  $BWDSTART = FALSE
  LDAT_ACT = LCPDAT1
  FDAT_ACT = FP3
  BAS(#CP_PARAMS, 0.5)
  SET_CD_PARAMS (0)
  TRIGGER WHEN DISTANCE = 1 DELAY = ArcGetDelay(#PreDefinition, WDAT1) DO ArcMainNG(#PreDefinition, WDAT1, WP3) PRIO = -1
  TRIGGER WHEN PATH = ArcGetPath(#OnTheFlyArcOn, WDAT1) DELAY = ArcGetDelay(#GasPreflow, WDAT1) DO ArcMainNG(#GasPreflow, WDAT1, WP3) PRIO = -1
  TRIGGER WHEN PATH = ArcGetPath(#OnTheFlyArcOn, WDAT1) DELAY = 0 DO ArcMainNG(#ArcOnMoveStd, WDAT1, WP3) PRIO = -1
  ArcMainNG(#ArcOnBeforeMoveStd, WDAT1, WP3)
  LIN XP3
  ArcMainNG(#ArcOnAfterMoveStd, WDAT1, WP3)
;ENDFOLD
   $VEL.CP = 0.060
   LIN  {X -2.694, Y 7.487, Z 19.900, A 0.000, B 0.000, C 0.000} C_DIS

;FOLD ARCOFF WDAT2 LIN P4 CPDAT2 Tool[1]:cmttorch Base[1]:vrashatel ;%{PE}
  ;FOLD Parameters ;%{h}
    ;Params IlfProvider=kukaroboter.arctech.arcofflin; Kuka.IsGlobalPoint=False; Kuka.PointName=P4; Kuka.BlendingEnabled=False; Kuka.MoveDataName=CPDAT2; Kuka.VelocityPath=0.01; Kuka.CurrentCDSetIndex=0; Kuka.MovementParameterFieldEnabled=True; ArcTech.WdatVarName=WDAT2; ArcTech.Basic=3.4.3.1264
  ;ENDFOLD
  $BWDSTART = FALSE
  LDAT_ACT = LCPDAT2
  FDAT_ACT = FP4
  BAS(#CP_PARAMS, gArcBasVelDefinition)
  SET_CD_PARAMS (0)
  TRIGGER WHEN PATH = ArcGetPath(#ArcOffBefore, WDAT2) DELAY = 0 DO ArcMainNG(#ArcOffBeforeOffStd, WDAT2, WP4) PRIO = -1
  TRIGGER WHEN PATH = ArcGetPath(#OnTheFlyArcOff, WDAT2) DELAY = 0 DO ArcMainNG(#ArcOffMoveStd, WDAT2, WP4) PRIO = -1
  ArcMainNG(#ArcOffBeforeMoveStd, WDAT2, WP4)
  LIN XP4
  ArcMainNG(#ArcOffAfterMoveStd, WDAT2, WP4)
;ENDFOLD
   $VEL.CP = 0.080
   LIN  {X -2.129, Y 7.487, Z 19.900, A 0.000, B 0.000, C 0.000} C_DIS

;FOLD ARCON WDAT1 LIN P3 Vel=0.5 m/s CPDAT1 Tool[1]:cmttorch Base[1]:vrashatel ;%{PE}
  ;FOLD Parameters ;%{h}
    ;Params IlfProvider=kukaroboter.arctech.arconlin; Kuka.IsGlobalPoint=False; Kuka.PointName=P3; Kuka.BlendingEnabled=False; Kuka.MoveDataName=CPDAT1; Kuka.VelocityPath=0.5; Kuka.CurrentCDSetIndex=0; Kuka.MovementParameterFieldEnabled=True; ArcTech.WdatVarName=WDAT1; ArcTech.Basic=3.4.3.1264
  ;ENDFOLD
  $BWDSTART = FALSE
  LDAT_ACT = LCPDAT1
  FDAT_ACT = FP3
  BAS(#CP_PARAMS, 0.5)
  SET_CD_PARAMS (0)
  TRIGGER WHEN DISTANCE = 1 DELAY = ArcGetDelay(#PreDefinition, WDAT1) DO ArcMainNG(#PreDefinition, WDAT1, WP3) PRIO = -1
  TRIGGER WHEN PATH = ArcGetPath(#OnTheFlyArcOn, WDAT1) DELAY = ArcGetDelay(#GasPreflow, WDAT1) DO ArcMainNG(#GasPreflow, WDAT1, WP3) PRIO = -1
  TRIGGER WHEN PATH = ArcGetPath(#OnTheFlyArcOn, WDAT1) DELAY = 0 DO ArcMainNG(#ArcOnMoveStd, WDAT1, WP3) PRIO = -1
  ArcMainNG(#ArcOnBeforeMoveStd, WDAT1, WP3)
  LIN XP3
  ArcMainNG(#ArcOnAfterMoveStd, WDAT1, WP3)
;ENDFOLD
   $VEL.CP = 0.060
   LIN  {X -0.787, Y 8.829, Z 19.900, A 0.000, B 0.000, C 0.000} C_DIS

;FOLD ARCOFF WDAT2 LIN P4 CPDAT2 Tool[1]:cmttorch Base[1]:vrashatel ;%{PE}
  ;FOLD Parameters ;%{h}
    ;Params IlfProvider=kukaroboter.arctech.arcofflin; Kuka.IsGlobalPoint=False; Kuka.PointName=P4; Kuka.BlendingEnabled=False; Kuka.MoveDataName=CPDAT2; Kuka.VelocityPath=0.01; Kuka.CurrentCDSetIndex=0; Kuka.MovementParameterFieldEnabled=True; ArcTech.WdatVarName=WDAT2; ArcTech.Basic=3.4.3.1264
  ;ENDFOLD
  $BWDSTART = FALSE
  LDAT_ACT = LCPDAT2
  FDAT_ACT = FP4
  BAS(#CP_PARAMS, gArcBasVelDefinition)
  SET_CD_PARAMS (0)
  TRIGGER WHEN PATH = ArcGetPath(#ArcOffBefore, WDAT2) DELAY = 0 DO ArcMainNG(#ArcOffBeforeOffStd, WDAT2, WP4) PRIO = -1
  TRIGGER WHEN PATH = ArcGetPath(#OnTheFlyArcOff, WDAT2) DELAY = 0 DO ArcMainNG(#ArcOffMoveStd, WDAT2, WP4) PRIO = -1
  ArcMainNG(#ArcOffBeforeMoveStd, WDAT2, WP4)
  LIN XP4
  ArcMainNG(#ArcOffAfterMoveStd, WDAT2, WP4)
;ENDFOLD
   $VEL.CP = 0.080
   LIN  {X -0.221, Y 8.829, Z 19.900, A 0.000, B 0.000, C 0.000} C_DIS

;FOLD ARCON WDAT1 LIN P3 Vel=0.5 m/s CPDAT1 Tool[1]:cmttorch Base[1]:vrashatel ;%{PE}
  ;FOLD Parameters ;%{h}
    ;Params IlfProvider=kukaroboter.arctech.arconlin; Kuka.IsGlobalPoint=False; Kuka.PointName=P3; Kuka.BlendingEnabled=False; Kuka.MoveDataName=CPDAT1; Kuka.VelocityPath=0.5; Kuka.CurrentCDSetIndex=0; Kuka.MovementParameterFieldEnabled=True; ArcTech.WdatVarName=WDAT1; ArcTech.Basic=3.4.3.1264
  ;ENDFOLD
  $BWDSTART = FALSE
  LDAT_ACT = LCPDAT1
  FDAT_ACT = FP3
  BAS(#CP_PARAMS, 0.5)
  SET_CD_PARAMS (0)
  TRIGGER WHEN DISTANCE = 1 DELAY = ArcGetDelay(#PreDefinition, WDAT1) DO ArcMainNG(#PreDefinition, WDAT1, WP3) PRIO = -1
  TRIGGER WHEN PATH = ArcGetPath(#OnTheFlyArcOn, WDAT1) DELAY = ArcGetDelay(#GasPreflow, WDAT1) DO ArcMainNG(#GasPreflow, WDAT1, WP3) PRIO = -1
  TRIGGER WHEN PATH = ArcGetPath(#OnTheFlyArcOn, WDAT1) DELAY = 0 DO ArcMainNG(#ArcOnMoveStd, WDAT1, WP3) PRIO = -1
  ArcMainNG(#ArcOnBeforeMoveStd, WDAT1, WP3)
  LIN XP3
  ArcMainNG(#ArcOnAfterMoveStd, WDAT1, WP3)
;ENDFOLD
   $VEL.CP = 0.060
   LIN  {X -1.563, Y 7.487, Z 19.900, A 0.000, B 0.000, C 0.000} C_DIS

;FOLD ARCOFF WDAT2 LIN P4 CPDAT2 Tool[1]:cmttorch Base[1]:vrashatel ;%{PE}
  ;FOLD Parameters ;%{h}
    ;Params IlfProvider=kukaroboter.arctech.arcofflin; Kuka.IsGlobalPoint=False; Kuka.PointName=P4; Kuka.BlendingEnabled=False; Kuka.MoveDataName=CPDAT2; Kuka.VelocityPath=0.01; Kuka.CurrentCDSetIndex=0; Kuka.MovementParameterFieldEnabled=True; ArcTech.WdatVarName=WDAT2; ArcTech.Basic=3.4.3.1264
  ;ENDFOLD
  $BWDSTART = FALSE
  LDAT_ACT = LCPDAT2
  FDAT_ACT = FP4
  BAS(#CP_PARAMS, gArcBasVelDefinition)
  SET_CD_PARAMS (0)
  TRIGGER WHEN PATH = ArcGetPath(#ArcOffBefore, WDAT2) DELAY = 0 DO ArcMainNG(#ArcOffBeforeOffStd, WDAT2, WP4) PRIO = -1
  TRIGGER WHEN PATH = ArcGetPath(#OnTheFlyArcOff, WDAT2) DELAY = 0 DO ArcMainNG(#ArcOffMoveStd, WDAT2, WP4) PRIO = -1
  ArcMainNG(#ArcOffBeforeMoveStd, WDAT2, WP4)
  LIN XP4
  ArcMainNG(#ArcOffAfterMoveStd, WDAT2, WP4)
;ENDFOLD
   $VEL.CP = 0.080
   LIN  {X -0.997, Y 7.487, Z 19.900, A 0.000, B 0.000, C 0.000} C_DIS

;FOLD ARCON WDAT1 LIN P3 Vel=0.5 m/s CPDAT1 Tool[1]:cmttorch Base[1]:vrashatel ;%{PE}
  ;FOLD Parameters ;%{h}
    ;Params IlfProvider=kukaroboter.arctech.arconlin; Kuka.IsGlobalPoint=False; Kuka.PointName=P3; Kuka.BlendingEnabled=False; Kuka.MoveDataName=CPDAT1; Kuka.VelocityPath=0.5; Kuka.CurrentCDSetIndex=0; Kuka.MovementParameterFieldEnabled=True; ArcTech.WdatVarName=WDAT1; ArcTech.Basic=3.4.3.1264
  ;ENDFOLD
  $BWDSTART = FALSE
  LDAT_ACT = LCPDAT1
  FDAT_ACT = FP3
  BAS(#CP_PARAMS, 0.5)
  SET_CD_PARAMS (0)
  TRIGGER WHEN DISTANCE = 1 DELAY = ArcGetDelay(#PreDefinition, WDAT1) DO ArcMainNG(#PreDefinition, WDAT1, WP3) PRIO = -1
  TRIGGER WHEN PATH = ArcGetPath(#OnTheFlyArcOn, WDAT1) DELAY = ArcGetDelay(#GasPreflow, WDAT1) DO ArcMainNG(#GasPreflow, WDAT1, WP3) PRIO = -1
  TRIGGER WHEN PATH = ArcGetPath(#OnTheFlyArcOn, WDAT1) DELAY = 0 DO ArcMainNG(#ArcOnMoveStd, WDAT1, WP3) PRIO = -1
  ArcMainNG(#ArcOnBeforeMoveStd, WDAT1, WP3)
  LIN XP3
  ArcMainNG(#ArcOnAfterMoveStd, WDAT1, WP3)
;ENDFOLD
   $VEL.CP = 0.060
   LIN  {X 0.344, Y 8.829, Z 19.900, A 0.000, B 0.000, C 0.000} C_DIS

;FOLD ARCOFF WDAT2 LIN P4 CPDAT2 Tool[1]:cmttorch Base[1]:vrashatel ;%{PE}
  ;FOLD Parameters ;%{h}
    ;Params IlfProvider=kukaroboter.arctech.arcofflin; Kuka.IsGlobalPoint=False; Kuka.PointName=P4; Kuka.BlendingEnabled=False; Kuka.MoveDataName=CPDAT2; Kuka.VelocityPath=0.01; Kuka.CurrentCDSetIndex=0; Kuka.MovementParameterFieldEnabled=True; ArcTech.WdatVarName=WDAT2; ArcTech.Basic=3.4.3.1264
  ;ENDFOLD
  $BWDSTART = FALSE
  LDAT_ACT = LCPDAT2
  FDAT_ACT = FP4
  BAS(#CP_PARAMS, gArcBasVelDefinition)
  SET_CD_PARAMS (0)
  TRIGGER WHEN PATH = ArcGetPath(#ArcOffBefore, WDAT2) DELAY = 0 DO ArcMainNG(#ArcOffBeforeOffStd, WDAT2, WP4) PRIO = -1
  TRIGGER WHEN PATH = ArcGetPath(#OnTheFlyArcOff, WDAT2) DELAY = 0 DO ArcMainNG(#ArcOffMoveStd, WDAT2, WP4) PRIO = -1
  ArcMainNG(#ArcOffBeforeMoveStd, WDAT2, WP4)
  LIN XP4
  ArcMainNG(#ArcOffAfterMoveStd, WDAT2, WP4)
;ENDFOLD
   $VEL.CP = 0.080
   LIN  {X 0.910, Y 8.829, Z 19.900, A 0.000, B 0.000, C 0.000} C_DIS

;FOLD ARCON WDAT1 LIN P3 Vel=0.5 m/s CPDAT1 Tool[1]:cmttorch Base[1]:vrashatel ;%{PE}
  ;FOLD Parameters ;%{h}
    ;Params IlfProvider=kukaroboter.arctech.arconlin; Kuka.IsGlobalPoint=False; Kuka.PointName=P3; Kuka.BlendingEnabled=False; Kuka.MoveDataName=CPDAT1; Kuka.VelocityPath=0.5; Kuka.CurrentCDSetIndex=0; Kuka.MovementParameterFieldEnabled=True; ArcTech.WdatVarName=WDAT1; ArcTech.Basic=3.4.3.1264
  ;ENDFOLD
  $BWDSTART = FALSE
  LDAT_ACT = LCPDAT1
  FDAT_ACT = FP3
  BAS(#CP_PARAMS, 0.5)
  SET_CD_PARAMS (0)
  TRIGGER WHEN DISTANCE = 1 DELAY = ArcGetDelay(#PreDefinition, WDAT1) DO ArcMainNG(#PreDefinition, WDAT1, WP3) PRIO = -1
  TRIGGER WHEN PATH = ArcGetPath(#OnTheFlyArcOn, WDAT1) DELAY = ArcGetDelay(#GasPreflow, WDAT1) DO ArcMainNG(#GasPreflow, WDAT1, WP3) PRIO = -1
  TRIGGER WHEN PATH = ArcGetPath(#OnTheFlyArcOn, WDAT1) DELAY = 0 DO ArcMainNG(#ArcOnMoveStd, WDAT1, WP3) PRIO = -1
  ArcMainNG(#ArcOnBeforeMoveStd, WDAT1, WP3)
  LIN XP3
  ArcMainNG(#ArcOnAfterMoveStd, WDAT1, WP3)
;ENDFOLD
   $VEL.CP = 0.060
   LIN  {X -0.432, Y 7.487, Z 19.900, A 0.000, B 0.000, C 0.000} C_DIS

;FOLD ARCOFF WDAT2 LIN P4 CPDAT2 Tool[1]:cmttorch Base[1]:vrashatel ;%{PE}
  ;FOLD Parameters ;%{h}
    ;Params IlfProvider=kukaroboter.arctech.arcofflin; Kuka.IsGlobalPoint=False; Kuka.PointName=P4; Kuka.BlendingEnabled=False; Kuka.MoveDataName=CPDAT2; Kuka.VelocityPath=0.01; Kuka.CurrentCDSetIndex=0; Kuka.MovementParameterFieldEnabled=True; ArcTech.WdatVarName=WDAT2; ArcTech.Basic=3.4.3.1264
  ;ENDFOLD
  $BWDSTART = FALSE
  LDAT_ACT = LCPDAT2
  FDAT_ACT = FP4
  BAS(#CP_PARAMS, gArcBasVelDefinition)
  SET_CD_PARAMS (0)
  TRIGGER WHEN PATH = ArcGetPath(#ArcOffBefore, WDAT2) DELAY = 0 DO ArcMainNG(#ArcOffBeforeOffStd, WDAT2, WP4) PRIO = -1
  TRIGGER WHEN PATH = ArcGetPath(#OnTheFlyArcOff, WDAT2) DELAY = 0 DO ArcMainNG(#ArcOffMoveStd, WDAT2, WP4) PRIO = -1
  ArcMainNG(#ArcOffBeforeMoveStd, WDAT2, WP4)
  LIN XP4
  ArcMainNG(#ArcOffAfterMoveStd, WDAT2, WP4)
;ENDFOLD
   $VEL.CP = 0.080
   LIN  {X 0.133, Y 7.487, Z 19.900, A 0.000, B 0.000, C 0.000} C_DIS

;FOLD ARCON WDAT1 LIN P3 Vel=0.5 m/s CPDAT1 Tool[1]:cmttorch Base[1]:vrashatel ;%{PE}
  ;FOLD Parameters ;%{h}
    ;Params IlfProvider=kukaroboter.arctech.arconlin; Kuka.IsGlobalPoint=False; Kuka.PointName=P3; Kuka.BlendingEnabled=False; Kuka.MoveDataName=CPDAT1; Kuka.VelocityPath=0.5; Kuka.CurrentCDSetIndex=0; Kuka.MovementParameterFieldEnabled=True; ArcTech.WdatVarName=WDAT1; ArcTech.Basic=3.4.3.1264
  ;ENDFOLD
  $BWDSTART = FALSE
  LDAT_ACT = LCPDAT1
  FDAT_ACT = FP3
  BAS(#CP_PARAMS, 0.5)
  SET_CD_PARAMS (0)
  TRIGGER WHEN DISTANCE = 1 DELAY = ArcGetDelay(#PreDefinition, WDAT1) DO ArcMainNG(#PreDefinition, WDAT1, WP3) PRIO = -1
  TRIGGER WHEN PATH = ArcGetPath(#OnTheFlyArcOn, WDAT1) DELAY = ArcGetDelay(#GasPreflow, WDAT1) DO ArcMainNG(#GasPreflow, WDAT1, WP3) PRIO = -1
  TRIGGER WHEN PATH = ArcGetPath(#OnTheFlyArcOn, WDAT1) DELAY = 0 DO ArcMainNG(#ArcOnMoveStd, WDAT1, WP3) PRIO = -1
  ArcMainNG(#ArcOnBeforeMoveStd, WDAT1, WP3)
  LIN XP3
  ArcMainNG(#ArcOnAfterMoveStd, WDAT1, WP3)
;ENDFOLD
   $VEL.CP = 0.060
   LIN  {X 1.475, Y 8.829, Z 19.900, A 0.000, B 0.000, C 0.000} C_DIS

;FOLD ARCOFF WDAT2 LIN P4 CPDAT2 Tool[1]:cmttorch Base[1]:vrashatel ;%{PE}
  ;FOLD Parameters ;%{h}
    ;Params IlfProvider=kukaroboter.arctech.arcofflin; Kuka.IsGlobalPoint=False; Kuka.PointName=P4; Kuka.BlendingEnabled=False; Kuka.MoveDataName=CPDAT2; Kuka.VelocityPath=0.01; Kuka.CurrentCDSetIndex=0; Kuka.MovementParameterFieldEnabled=True; ArcTech.WdatVarName=WDAT2; ArcTech.Basic=3.4.3.1264
  ;ENDFOLD
  $BWDSTART = FALSE
  LDAT_ACT = LCPDAT2
  FDAT_ACT = FP4
  BAS(#CP_PARAMS, gArcBasVelDefinition)
  SET_CD_PARAMS (0)
  TRIGGER WHEN PATH = ArcGetPath(#ArcOffBefore, WDAT2) DELAY = 0 DO ArcMainNG(#ArcOffBeforeOffStd, WDAT2, WP4) PRIO = -1
  TRIGGER WHEN PATH = ArcGetPath(#OnTheFlyArcOff, WDAT2) DELAY = 0 DO ArcMainNG(#ArcOffMoveStd, WDAT2, WP4) PRIO = -1
  ArcMainNG(#ArcOffBeforeMoveStd, WDAT2, WP4)
  LIN XP4
  ArcMainNG(#ArcOffAfterMoveStd, WDAT2, WP4)
;ENDFOLD
   $VEL.CP = 0.080
   LIN  {X 2.041, Y 8.829, Z 19.900, A 0.000, B 0.000, C 0.000} C_DIS

;FOLD ARCON WDAT1 LIN P3 Vel=0.5 m/s CPDAT1 Tool[1]:cmttorch Base[1]:vrashatel ;%{PE}
  ;FOLD Parameters ;%{h}
    ;Params IlfProvider=kukaroboter.arctech.arconlin; Kuka.IsGlobalPoint=False; Kuka.PointName=P3; Kuka.BlendingEnabled=False; Kuka.MoveDataName=CPDAT1; Kuka.VelocityPath=0.5; Kuka.CurrentCDSetIndex=0; Kuka.MovementParameterFieldEnabled=True; ArcTech.WdatVarName=WDAT1; ArcTech.Basic=3.4.3.1264
  ;ENDFOLD
  $BWDSTART = FALSE
  LDAT_ACT = LCPDAT1
  FDAT_ACT = FP3
  BAS(#CP_PARAMS, 0.5)
  SET_CD_PARAMS (0)
  TRIGGER WHEN DISTANCE = 1 DELAY = ArcGetDelay(#PreDefinition, WDAT1) DO ArcMainNG(#PreDefinition, WDAT1, WP3) PRIO = -1
  TRIGGER WHEN PATH = ArcGetPath(#OnTheFlyArcOn, WDAT1) DELAY = ArcGetDelay(#GasPreflow, WDAT1) DO ArcMainNG(#GasPreflow, WDAT1, WP3) PRIO = -1
  TRIGGER WHEN PATH = ArcGetPath(#OnTheFlyArcOn, WDAT1) DELAY = 0 DO ArcMainNG(#ArcOnMoveStd, WDAT1, WP3) PRIO = -1
  ArcMainNG(#ArcOnBeforeMoveStd, WDAT1, WP3)
  LIN XP3
  ArcMainNG(#ArcOnAfterMoveStd, WDAT1, WP3)
;ENDFOLD
   $VEL.CP = 0.060
   LIN  {X 0.699, Y 7.487, Z 19.900, A 0.000, B 0.000, C 0.000} C_DIS

;FOLD ARCOFF WDAT2 LIN P4 CPDAT2 Tool[1]:cmttorch Base[1]:vrashatel ;%{PE}
  ;FOLD Parameters ;%{h}
    ;Params IlfProvider=kukaroboter.arctech.arcofflin; Kuka.IsGlobalPoint=False; Kuka.PointName=P4; Kuka.BlendingEnabled=False; Kuka.MoveDataName=CPDAT2; Kuka.VelocityPath=0.01; Kuka.CurrentCDSetIndex=0; Kuka.MovementParameterFieldEnabled=True; ArcTech.WdatVarName=WDAT2; ArcTech.Basic=3.4.3.1264
  ;ENDFOLD
  $BWDSTART = FALSE
  LDAT_ACT = LCPDAT2
  FDAT_ACT = FP4
  BAS(#CP_PARAMS, gArcBasVelDefinition)
  SET_CD_PARAMS (0)
  TRIGGER WHEN PATH = ArcGetPath(#ArcOffBefore, WDAT2) DELAY = 0 DO ArcMainNG(#ArcOffBeforeOffStd, WDAT2, WP4) PRIO = -1
  TRIGGER WHEN PATH = ArcGetPath(#OnTheFlyArcOff, WDAT2) DELAY = 0 DO ArcMainNG(#ArcOffMoveStd, WDAT2, WP4) PRIO = -1
  ArcMainNG(#ArcOffBeforeMoveStd, WDAT2, WP4)
  LIN XP4
  ArcMainNG(#ArcOffAfterMoveStd, WDAT2, WP4)
;ENDFOLD
   $VEL.CP = 0.080
   LIN  {X 1.265, Y 7.487, Z 19.900, A 0.000, B 0.000, C 0.000} C_DIS

